# B&R Automation Studio project 305841_E00002_0 (part 11)

#### GAProcIO.fun - Exported functions and function blocks
```iecst
(********************************************************************
 * COPYRIGHT -- General Atomics
 ********************************************************************
 * Library: GAProcIO
 * File: GAProcIO.fun
 * Author: Administrator
 * Created: September 11, 2015
 ********************************************************************
 * Functions and function blocks of library GAAnalog
 ********************************************************************)

FUNCTION_BLOCK fbSclAlmAI (* Scale analog input and process alarms using the reference parameters *)
	VAR_INPUT
		_InInputStruct : REFERENCE TO sAnalogInput; (* structure representing the analog input to scale *)
		_InParamsStruct : REFERENCE TO sAnalogInputParams; (* structure representing the analog parameters *)
		_InSentinel : REAL; (* value to use if signal is invalid *) (* Set the scaling params and alm timer delays upon rising edge *) (* Must go low and high again to set again *)
		_InSetParams : BOOL := FALSE;
	END_VAR
	VAR
		SetParamsOS : BOOL := FALSE; (* set parameters one-shot *)
		rawAdj : REAL;
		almsRaw : UDINT; (* non-time delayed alarms *) (* deadband values, calculated from EU range and db pct *) (* pvs must rise above threshold by the corresponding value in order to be considered clear *)
		almRangeLoDbVal : REAL;
		almRangeHiDbVal : REAL;
		almLoLoDbVal : REAL;
		almLoDbVal : REAL; (* pvs must drop below threshold by the corresponding value in order to be considered clear *)
		almHiDbVal : REAL;
		almHiHiDbVal : REAL; (* alarm timers *)
		tmrAlmRangeLoOn : TON; (* on delay timers *)
		tmrAlmLoLoOn : TON;
		tmrAlmLoOn : TON;
		tmrAlmRangeHiOn : TON;
		tmrAlmHiOn : TON;
		tmrAlmHiHiOn : TON;
		tmrAlmRangeLoOff : TOF; (* off delay timers *)
		tmrAlmLoLoOff : TOF;
		tmrAlmLoOff : TOF;
		tmrAlmRangeHiOff : TOF;
		tmrAlmHiOff : TOF;
		tmrAlmHiHiOff : TOF;
		fbNoiseFilter : fbLpFilter; (* filter the scaled value *)
	END_VAR
END_FUNCTION_BLOCK

FUNCTION_BLOCK fbLpFilter (* Low pass filter *)
	VAR_INPUT
		_InPassThru : BOOL := FALSE; (* filter coefficient *) (* Value between 0 and 1, not inclusive of 1. *) (* K=0 no filtering, K=0.9999 lots of filtering *)
		_InK : REAL := 0.0;
		_InVal : REAL; (* input value *)
	END_VAR
	VAR_OUTPUT
		_OutFilteredVal : REAL; (* filtered value output  *)
	END_VAR
	VAR
		lastOut : REAL;
		firstScanOS : BOOL := FALSE;
		KChecked : REAL := 0.0;
	END_VAR
END_FUNCTION_BLOCK

FUNCTION_BLOCK fbProcDI (* process DI *)
	VAR_INPUT
		_InInputStruct : REFERENCE TO sDigitalInput; (* structure representing the digital input to process *)
		_InParamsStruct : REFERENCE TO sDigitalInputParams; (* structure representing the digital input parameters *)
		_InSentinel : BOOL := FALSE; (* value to use if signal is invalid *) (* Set the params and alm timer delays upon rising edge *) (* Must go low and high again to set again *)
		_InSetParams : BOOL := FALSE;
	END_VAR
	VAR
		SetParamsOS : BOOL := FALSE; (* set parameters one-shot *)
    value : BOOL;
    valueDly : BOOL;
    almsRaw : UDINT;
    prevParams : sDigitalInputParams; (* previous params -- used for auto param update *)
    paramSize : UDINT := 0;
    cmpResult : DINT;
		tmrOn : TON;
		tmrAlmLoOn : TON;
		tmrAlmHiOn : TON;
		tmrOff : TOF; (* non-time delayed alarms *)
		tmrAlmLoOff : TOF;
		tmrAlmHiOff : TOF;
	END_VAR
END_FUNCTION_BLOCK

FUNCTION_BLOCK fbProcPB
	VAR_INPUT
    _InPBIn : BOOL := FALSE;
    _InPBClear : BOOL := FALSE; (* Force state to be cleared *)
		_InPBType : eGAPIO_PB_BEHAVIOR_TYPE := GAPIO_PBBT_MOMENTARY;
		_InPulseTime : TIME := T#500ms;
	END_VAR
	VAR_OUTPUT
		_OutState : BOOL := FALSE;
	END_VAR
	VAR
		pressOS : BOOL := FALSE;
		state : BOOL := FALSE;
		tmrPulse : TON;
	END_VAR
END_FUNCTION_BLOCK
```

### Library Logical/Libraries/GAMpMotion (IEC) - Mapp Motion Helper Functions

#### Types.typ
```iecst
TYPE
  eGAMOT_HOME_FB_STATUS :
    (
    GAMOT_HMFBS_NOT_ACTIVE := 0,
    GAMOT_HMFBS_ENABLED := 1,
    GAMOT_HMFBS_HOMING := 2,
    GAMOT_HMFBS_HOMED := 3,
    GAMOT_HMFBS_ERR_START_STATE := -1, (* must be in disabled or standstill to start *)
    GAMOT_HMFBS_ERR_HOMING := -2 (* error occured during homing *)
  ) := GAMOT_HMFBS_NOT_ACTIVE;

  eGAMOT_AXIS_STATE_MACHINE_STATE :
    (
    (* axis state constants *)
    (* states which dont't issue move commands *)
    GAMOT_ASMS_INITIAL := 0, (*constant for an undefined state. Also used for initial state *)
    GAMOT_ASMS_IGNORE := 1, (*constant for ignore state *)
    GAMOT_ASMS_VALID_CHECK := 2, (*constant for invalid state *)
    GAMOT_ASMS_DISABLED := 3, (*constant for the disabled state *)
    GAMOT_ASMS_ENABLED := 4, (*constant for a waiting while powered *)
    GAMOT_ASMS_HOME_REQ := 5, (*constant for the state in which the axis home was requested *)
    GAMOT_ASMS_HOMING := 6, (*constant for the state in which the axis is being referenced *)
    GAMOT_ASMS_HOMED := 7, (*constant for the state in which the axis is referenced *)
    GAMOT_ASMS_CHK_RESTORE_POS := 8, (* constant for Init Endless Position State *)
    GAMOT_ASMS_RESTORE_POS := 9, (* constant for Init Endless Position Error State *)
    GAMOT_ASMS_ERROR_STOP := 10, (*constant for function block error stop state *)
    GAMOT_ASMS_ERROR_DRVRSTWAIT := 11, (*constant for axis error drive reset wait state *)
    GAMOT_ASMS_ERROR_DISABLE := 12, (*constant for axis error drive reset wait state *)
    GAMOT_ASMS_ERROR_DRVRST:= 13, (*constant for axis error drive reset state *)
    (* states which are stop moves *)
    GAMOT_ASMS_HALT := 20, (*constant for the state in which motion is halted *)
    GAMOT_ASMS_STOP := 21, (*constant for the state in which motion is stopped, awaiting stop reset req *)
    GAMOT_ASMS_STOP_RESET := 22, (*constant for the state in which movements are stopped after stop reset req received *)
    GAMOT_ASMS_HALT_DISABLE := 23, (* constant for the state which stops the axes before disabling *)
    (* states which are velocity  moves *)
    GAMOT_ASMS_JOG := 31, (*constant for the state in which jogging movement is executed *)
    GAMOT_ASMS_JOGPOSLIMIT := 32, (*constant for the state in which jogging positive limit movement is executed *)
    GAMOT_ASMS_JOGNEGLIMIT := 33, (*constant for the state in which jogging positive limit movement is executed *)
    (* states which are velocity moves *)
    GAMOT_ASMS_MOVE_VELOCITY := 41, (* constant for the state in which a movement with a defined velocity is executed *)
    (* states which are relative moves *)
    GAMOT_ASMS_MOVE_RELATIVE := 51, (*constant for the state in which a movement with defined distance is executed*)
    (* states which are absolute moves *)
    GAMOT_ASMS_MOVE_ABSOLUTE := 61, (*constant for the state in which a movement to defined position is executed *)
    (* states related to coordinated moves *)
    GAMOT_ASMS_ENGAGED_AS_SLAVE := 71, (* geared or cammed to a master axis (coordinated slave) *)
    GAMOT_ASMS_DISENGAGE_AS_SLAVE := 72 (* disengaging from a master axis (coordinated slave) *)
  ) := GAMOT_ASMS_INITIAL;

  eGAMOT_MOVE_DESIGNATION :
    ( (* Move Designation *)
    (* Be careful about changing values -- HMI ramifications *)
    (* Values support bit packed int *)
    GAMOT_MD_UNKNOWN                := -1, (* no HMI selection *)
    GAMOT_MD_NO_MOVE_COMMANDED      := 16#00,
    GAMOT_MD_JOG_VELOCITY_UP_FWD    := 16#01,
    GAMOT_MD_JOG_VELOCITY_DOWN_REV  := 16#02,
    GAMOT_MD_JOG_LIMIT_UP_FWD       := 16#04,
    GAMOT_MD_JOG_LIMIT_DOWN_REV     := 16#08,
    GAMOT_MD_VELOCITY               := 16#10,
    GAMOT_MD_RELATIVE               := 16#20,
    GAMOT_MD_ABSOLUTE               := 16#40,
    GAMOT_MD_COORDINATED            := 16#80
  ) := GAMOT_MD_NO_MOVE_COMMANDED;

  sMot_PositionLimits : STRUCT (* axis travel limits. *)
    (* This is a separate structure from move params so instances can
    efficiently be made permanent variables *)
    PositionLimitPos : LREAL;
    PositionLimitNeg : LREAL;
  END_STRUCT;

  sMot_HmiAxisReqs : STRUCT
    (* Move or motion related requests *)
    (* NOTE: BE CAREFUL about changes and reordering -- HMI and memcopy/memset ramifications *)
    (* Boolean reqs are cleared with memset so adding/removing/moving may be problematic *)
    (* NOTE: Do not add bool reqs before moveReq that should be cleared while in safe/emo modes. *)
    _beginResetSection : BOOL := FALSE;
    moveReq : BOOL := FALSE;
    haltReq : BOOL := FALSE;
    stopReq : BOOL := FALSE;
    homeSetZeroReq : BOOL := FALSE;
    homeSetOffsetReq : BOOL := FALSE;
    homeSetPosReq : BOOL := FALSE;
    enableReq : BOOL := FALSE;
    disableReq : BOOL := FALSE;
    manBrakeRelReq : BOOL := FALSE;
    clearManBrakeRelReq : BOOL := FALSE;
    offsetShiftReq : BOOL := FALSE; (* shift slave pos on the slave axis, shift value in slave units *)
    offsetShiftToMasterPosReq : BOOL := FALSE; (* shift slave position by axis offset in slave units *)
    phaseShiftReq : BOOL := FALSE; (* shift master pos on the slave axis, shift value in master units *)
    gearInReq : BOOL := FALSE;
    camInReq : BOOL := FALSE;
    disengageSlaveReq : BOOL := FALSE; (* Disengage cam and gear *)
    _endResetSection : BOOL := FALSE;
    (* NOTE: Do not add bool reqs after disengageSlaveReq that should be cleared in safe/emo modes.  HMI and memcopy/memset ramifications. *)
    (* Other requests *)
    (* NOTE: Do not add bool reqs before setPositionLimitsReq that should be cleared while in emo mode. *)
    (* Separate the below requests after disengageSlaveReq so they can be considered while in safe mode. *)
    (* These are things that can be done while in safe mode, but the ones above are cleared while in safe.*)
    setPositionLimitsReq : BOOL := FALSE;
    stopResetReq : BOOL := FALSE;
    errorResetReq : BOOL := FALSE;
    driveResetReq : BOOL := FALSE;
    axisNo : USINT := 0; (* convenience axis number this structure corresponds to *)
    (* gear in related *)
    gearRatioNumerator : DINT := 1000; (* gear factor of the slave / measurment resolution of the slave *)
    gearRatioDenominator : DINT := 1000; (* gear factor of the master / measurment resolution of the master *)
    (* shift related *)
    shiftOverMasterDistance : BOOL := FALSE; (* H: Perofrm shift over specified master distance Use mcPROFBASE_MASTER_DISTANCE and shiftProfileDistance *)
    shiftType : SINT := 0; (* based on HMI radio buttons. 0: Relative, 1: Abs *)
    shiftDistance : LREAL := 0.0; (* phase/offset shift distance *)
    shiftProfileDistance : LREAL := 0.0; (* distance master moves during a shift *)
    (* cam related *)
    camId : UINT;
    camMasterOffset : LREAL := 0.0; (* gear factor of the slave / measurment resolution of the slave *)
    camSlaveOffset : LREAL := 0.0; (* gear factor of the master / measurment resolution of the master *)
    homePosition : LREAL := 0.0;
    positionLimits : sMot_PositionLimits;
    moveDesignation : eGAMOT_MOVE_DESIGNATION := GAMOT_MD_NO_MOVE_COMMANDED;
    (* HMI move req *)
    (* BE CAREFUL ABOUT MOVING/DELETING/ADDING/CHANGING MEMORY between Direction and MaxJerk *)
    (* MAY NEED TO ADJUST fgProcessHmiMoveReq instruction in GaMpMotion library *)
    (* These move params are copied to/from the HMI move req structure using memcpy *)
    _startParamCopy : BOOL := FALSE;
    Direction : McDirectionEnum := mcDIR_UNDEFINED; (* direction for commanded movements*)
    Distance : LREAL := 0.0; (* distance for move Commands *)
    Position : LREAL := 0.0; (* target position for home or the motion *)
    Velocity : REAL := 0.0; (* velocity for move Commands *)
    Acceleration : REAL := 1.0; (* acceleration for commanded movements *)
    Deceleration : REAL := 1.0; (* deceleration for commanded movements *)
    MaxJerk : REAL := 0.0; (* deceleration for commanded movements *)
    _endParamCopy : BOOL := FALSE;
    (* NOTE: BE CAREFUL ABOUT MOVING/DELETING/ADDING/CHANGING MEMORY between direction and MaxJerk *)
  END_STRUCT;

  sMot_PermissiveCheck : 	STRUCT (* used to halt/stop if out of allowable range or due to permissive *)
    (* 24 byte structure *)
    PermissiveHaltNeg : BOOL; (* byte 0 *)
    PermissiveHaltPos : BOOL; (* byte 1 *)
    CheckFailed : BOOL; (* byte 2 *)
    RangeLimitNeg : BOOL; (* byte 3 *)
    RangeLimitPos : BOOL; (* byte 4 *)
    spareBytes : ARRAY[0..2] OF BYTE; (* bytes 5-7 *)
    StartPosition : LREAL; (* byte 8-15 *)
    EstStoppingDistance : LREAL; (* byte 16-23 *)
  END_STRUCT;

  sMot_AxisStatus : 	STRUCT  (* drive state structure from MC_ReadStatus *)
    (* MpAxisBasic related *)
    IsCommuncationReady : BOOL := FALSE; (* MpAxisBasic is ready to communicate *)
    IsReadyToPowerOn : BOOL := FALSE; (* MpAxisBasic is ready for operation *)
    (* digital input status *)
    IsAtHomingSwitch : BOOL := FALSE;
    IsAtPositiveLimitSwitch : BOOL := FALSE;
    IsAtNegativeLimitSwitch : BOOL := FALSE;
    IsTrigger1Active : BOOL := FALSE;
    IsTrigger2Active : BOOL := FALSE;
    IsDriveEnableActive : BOOL := FALSE;
    (* general status *)
    IsInSimulation : BOOL := FALSE; (* Axis is operating in simulaiton mode *)
    IsPoweredOn : BOOL := FALSE;  (* axis is swtiched on/enabled *)
    IsTorqueLimitReady : BOOL := FALSE;
    IsBrakeManuallyReleased : BOOL := FALSE;
    IsHomed : BOOL := FALSE; (* axis is referenced *)
    IsJogging : BOOL := FALSE; (* performing movement *)
    IsAtJogLimit : BOOL := FALSE; (* the axis has reached one of two position limits *)
    IsAtTorqueLimit : BOOL := FALSE; (* the axis limit is active *)
    IsInVelocity : BOOL := FALSE; (* axis is running with a defined velocity *)
    IsInPosition : BOOL := FALSE; (* axis has acheived the desired position *)
    IsMoveActive : BOOL := FALSE; (* movement is active *)
    IsMoveDone : BOOL := FALSE; (* move complete *)
    IsStopped : BOOL := FALSE; (* axis is stopped *)
    (* auto-tune related *)
    IsAutoTuneDone : BOOL := FALSE;
    AutoTuneQuality : REAL := 0.0;
    (* general status values and structures *)
    SafeMotionDiagCode : UINT; (* from Safety Controller safe motion instruction *)
    Velocity : REAL:= INVALID_SENTINEL_REAL; (* actual axis velocity *)
    Position : LREAL:= INVALID_SENTINEL_LREAL; (* actual axis position. Includes MOD to keep value within a period value *)
    DrivePosition : LREAL := INVALID_SENTINEL_LREAL; (* actual axis position. Does not includes MOD so period is ignored *)
    CalculatedPosition1 : LREAL:= INVALID_SENTINEL_LREAL; (* calculated position -- axis specific *)
    CalculatedPosition2 : LREAL:= INVALID_SENTINEL_LREAL; (* calculated position -- axis specific *)
    CalculatedPosition3 : LREAL:= INVALID_SENTINEL_LREAL; (* calculated position -- axis specific *)
    (* Values to see progress of a move *)
    MoveStartPos : LREAL := INVALID_SENTINEL_LREAL;
    MoveEndPos : LREAL := INVALID_SENTINEL_LREAL;
    MoveDistanceRemaining : LREAL := 0.0;
    MoveDistanceComplete : LREAL := 0.0;
    StartupCount : UDINT := 0; (* number of times the drive was started since last PLC start *)
    PlcOpenState : McAxisPLCopenStateEnum;
    networkCommState : McCommunicationStateEnum;
    AxisDiagnostics : MpAxisDiagExtType;
    LibraryInfo : McLibraryInfoType;
    (* coupling related *)
    HasCoordinatedSlave : BOOL := FALSE;
    IsGearInSync : BOOL := FALSE; (* slave is in sync with the master *)
    IsGearInCompensation : BOOL := FALSE; (* slave is in compensation with the master *)
    IsCamInSync : BOOL := FALSE; (* slave is in sync with the master *)
    IsCamEndOfProfile : BOOL := FALSE; (* Pulsed output indicating cyclic end of cam *)
    IsCoordOffsetShiftStarted : BOOL := FALSE;
    IsCoordOffsetShiftAttained : BOOL := FALSE;
    IsCoordPhaseShiftStarted : BOOL := FALSE;
    IsCoordPhaseShiftAttained : BOOL := FALSE;
    CamStatus : McCamInStatusEnum;
    CoordActualOffsetShift : LREAL := 0.0; (* current shift of the slave *)
    CoordActualPhaseShift : LREAL := 0.0; (* current shift of the master axis *)
  END_STRUCT;

  sMot_MoveParameters : 	STRUCT  (*parameter structure*)
    (* NOTE: BE CAREFUL about changes and reordering -- HMI and memcopy ramifications *)
    (* put the permissive stuff at the beginning, so the move parameter updates to the *)
    (* MpAxisBasic instruction deal with contiguous memory *)
    PosMovePermissive : BOOL := FALSE; (* byte 0 only allow forward moves when high *)
    NegMovePermissive : BOOL := FALSE; (* byte 1 only allow reverse moves when high *)
    EnableTorqueLimit : BOOL := FALSE; (* byte 2 Limit torque for accel/decel *)
    EnableTorqueLimitPrev : BOOL := FALSE;  (* byte 3 prev value to detect change *)
    HaltOnSlaveDisengage : BOOL := FALSE; (* byte 4 if set, issue a halt when axis is disengaged *)
    spareBytes5_7 : ARRAY[0..2] OF BYTE; (* bytes 5-7 *)
    PermissiveCheck : sMot_PermissiveCheck; (* 24 byte structure. bytes 8-31 permissive and range check bits *)
    VelocityMin : REAL := 0.001; (* bytes 32-35 min and max allowed velocity *)
    VelocityMax : REAL := 100.0; (* bytes 36-39 *)
    AccelMin : REAL := 0.001; (* bytes 40-43 min and max allowed acceleration *)
    AccelMax : REAL := 100.0; (* bytes 44-47 *)
    DecelMin : REAL := 0.001; (* bytes 48-51 min and max allowed deceleration *)
    DecelMax : REAL := 100.0; (* bytes 52-55 *)
    _beginHmiSection : BOOL := FALSE;
    (* HMI move req related *)
    (* BE CAREFUL ABOUT MOVING/DELETING/ADDING/CHANGING MEMORY between Direction and MaxJerk
    (* and between Direction to the end of the structure.*)
    (* MAY NEED TO ADJUST fgProcessHmiAxisReq instruction in GaMpMotion library *)
    (* These move params are copied to/from the HMI move req structure using memcpy *)
    (* use MC enum for direction *)
    (* mcPOSITIVE_DIR = 0, mcNEGATIVE_DIR = 1, mcDIR_SHORTEST_WAY = 3, mcDIR_UNDEFINED = 9, for other values, see docs *)
    Direction : McDirectionEnum := mcDIR_UNDEFINED; (* bytes 56-59 direction for commanded movements*)
    Distance : LREAL := 0.0; (* bytes 60-67 distance for move Commands*)
    Position : LREAL := 0.0; (* bytes 68-75 target position for the movement *)
    Velocity : REAL := 0.0; (* bytes 76-79 velocity for move Commands*)
    Acceleration : REAL := 1.0; (* bytes 80-83 acceleration for commanded movements*)
    Deceleration : REAL := 1.0; (* bytes 84-87 deceleration for commanded movements*)
    MaxJerk : REAL := 0.0; (* bytes 88-91 *)
    (* NOTE: BE CAREFUL ABOUT MOVING/DELETING/ADDING/CHANGING MEMORY between Direction and MaxJerk *)
    (* End Hmi Move Req *)
    _endHmiSection : BOOL := FALSE;
    HomeParams : MpAxisHomingType; (* parameters for referencing the axis*)
    JogParams : MpAxisJogType; (* parameters for jog command *)
    StopParams : MpAxisStopType; (* parameters for stop command *)
    TorqueLimitParams : MpAxisLimitLoadType; (* parameters for torque limit *)
    AutoTuneParams : MpAxisAutoTuneType; (* parameters for auto tuning *)
  END_STRUCT;

  sMot_CouplingParameters : 	STRUCT  (* coupling parameter structure*)
    CouplingPermissive : BOOL := FALSE; (* axis allowing itself to be coupled as a slave *)
    GearInReq : BOOL := FALSE; (* Set to request gear coupling *)
    GearOutReq : BOOL := FALSE; (* Set to request gear decoupling *)
    CamInReq : BOOL := FALSE; (* Set to request cam coupling *)
    CamOutReq : BOOL := FALSE; (* Set to request cam decoupling *)
    OffsetShiftReq : BOOL := FALSE;(* Generate an offset shift in the position of the slave on the slave axis *)
    PhaseShiftReq : BOOL := FALSE; (* Geneate a phase shift in the position of the master on the slave axis *)
    SlaveAxisNo : USINT := 0; (* default to 0 so setting a value can be detected *)
    (* CAUTION
    mem compare and mem copy are used for these values when dealing with run time value changes.
    Be very careful about where you add values. For example, changes to values in the gearin section will
    cause a gearin update *)
    (* Gear In params *)
    _beginGearInSection : BOOL := FALSE;
    GearInRatioNumerator : DINT := 1000; (* Gear factor of the slave / Measurement resolution of the slave *)
    GearInRatioDenominator : DINT:= 1000; (* Gear factor of the master / Measurement resolution of the master *)
    GearInMasterValueSource : McValueSrcEnum := mcVALUE_ACTUAL; (* Master position source *)
    GearInBufferMode : McBufferModeEnum := mcABORTING; (* mcABORTING is the only mode currently supported *)
    _endGearInSection : BOOL := FALSE;
    (* Offset / Phase shift params *)
    (* The values in the common section are common to gear in, cam, and shift *)
    _beginShiftCommonSection : BOOL := FALSE;
    ShiftAccelerationMax : REAL; (* if 0 limit for slave axis is used *)
    ShiftDecelerationMax : REAL; (* if 0 limit for slave axis is used *)
    ShiftJerk : REAL := 0.0; (* non zero only supported with McProfGen *)
    ShiftProfileBaseMaxVelocity : REAL := 0.0; (* also use for cam adv paramm vel. 0.0: use max velocity master axis *)
    _endShiftCommonSection : BOOL := FALSE;
    _beginShiftSection : BOOL := FALSE;
    ShiftMode : McShiftModeEnum;
    ShiftProfileBase : McProfileBaseEnum;
    Shift : LREAL; (* shift distance *)
    ShiftVelocityMax : REAL;
    ShiftProfileDistance : LREAL;
    (* Zone params used with profile base mcXxx_ZONE *)
    ShiftZoneStartPosition : LREAL;
    ShiftZoneEndPosition : LREAL;
    ShiftZonePeriod : LREAL := 0.0; (* 0: period defined for the profile base is used *)
    _endShiftSection : BOOL := FALSE;
    _beginCamInSection : BOOL := FALSE;
    CamIsPeriodic : BOOL := TRUE; (* H: cam is performed periodically, L: cam is performed once *)
    CamId : UINT := 1; (* cam id used with CamIn *)
    CamMasterOffset : LREAL := 0.0;
    CamSlaveOffset : LREAL := 0.0;
    CamScalingMaster : DINT := 1000; (* Cam scaling factor for master *)
    CamScalingSlave : DINT := 1000; (* Cam scaling factor for scaling *)
    CamStartMode : McCamStartModeEnum;
    CamMasterValueSource : McValueSrcEnum := mcVALUE_ACTUAL; (* Master position source *)
    CamBufferMode : McBufferModeEnum := mcABORTING; (* mcABORTING is thye only mode currently supported *)
    _endCamInSection : BOOL := FALSE;
  END_STRUCT;

  sMot_AxisCommands : 	STRUCT  (*command structure for single and master axes*)
    MoveNotAllowed : BOOL:= TRUE; (* set if a requested move is not allowed, clear upon good request *)
    PlcSafetyEnable : BOOL := FALSE; (* PLC logic enable of SafeMC, via safety controller *)
    UpdateMoveParams : BOOL := FALSE; (* used to control the update bit to McAxisBasic when move params change *)
    EnableReq : BOOL:= FALSE; (* request enabling (powering on) the controller. *)
    DisableReq : BOOL:= FALSE; (* request disabeling (powering off) the controller *)
    EnableCmd : BOOL:= FALSE; (* enable (power on) the controller. Power off on false *)
    ReleaseBrakeReq : BOOL:= FALSE; (* request brake release if motor is off *)
    ClearReleaseBrakeReq : BOOL:= FALSE; (* clear brake release req *)
    ReleaseBrakeCmd : BOOL:= FALSE; (* release brake if motor is off *)
    HomeReq : BOOL:= FALSE; (* request setting of the reference position *)
    HomeCmd : BOOL:= FALSE; (* set the reference position *)
    MoveJogReq : BOOL:= FALSE; (* request jog move as long as is set. Direction set by MoveParameter.Direction *)
    MoveJogCmd : BOOL:= FALSE; (* jog (move) as long as is set. Direction set by MoveParameter.Direction *)
    MoveJogPositiveReq : BOOL:= FALSE; (* request jog move as long as is set. Stop at the software position limit *)
    MoveJogPositiveCmd : BOOL:= FALSE; (* jog (move) as long as is set. Stop at the software position limit *)
    MoveJogNegativeReq : BOOL:= FALSE; (* request jog move as long as is set. Stop at the software position limit *)
    MoveJogNegativeCmd : BOOL:= FALSE; (* jog (move) as long as is set. Stop at the software position limit *)
    MoveVelocityReq : BOOL:= FALSE; (* request move at a defined velocity *)
    MoveVelocityCmd : BOOL:= FALSE; (* move at a defined velocity *)
    MoveRelativeReq : BOOL:= FALSE; (* request move of a defined distance*)
    MoveRelativeCmd : BOOL:= FALSE; (* move a defined distance *)
    MoveAbsoluteReq : BOOL:= FALSE; (* request move to a defined position *)
    MoveAbsoluteCmd : BOOL:= FALSE; (* move to a defined position *)
    StopReq : BOOL:= FALSE; (* reqeust stop every active movement on the axis as long as is set *)
    StopCmd : BOOL:= FALSE; (* stop every active movement on the axis as long as is set *)
    StopResetReq : BOOL:= FALSE; (* set high to get out of STOPPED state *)
    HaltReq : BOOL:= FALSE; (* request stop every active movement on the axis *)
    HaltCmd : BOOL:= FALSE; (* stop every active movement on the axis *)
    DriveResetReq : BOOL:= FALSE; (* request drive reset *)
    DriveResetCmd : BOOL:= FALSE; (* drive reset command *)
    ErrorResetReq : BOOL:= FALSE; (* Request exit from Error Reset Wait *)
  END_STRUCT;

(*
  sMot_Error : 	STRUCT  (*error structure
    FBError : BOOL; (*an error occurred in a FB
    AxisError : BOOL; (*an axis error has occurred
    AxisWarning : BOOL; (*an axis warning has occurred
    AxisErrorStop : BOOL; (*axis is in ErrorStop state
    AcknowledgeAllReq : BOOL; (*user alarm acknowledge - ack all alarms
    AcknowledgeReq : BOOL; (*user alarm acknowledge
    AxisErrorCount : UINT; (*number of active axis errors
    AxisWarningCount : UINT; (*number of active axis warinings
    FBErrorCount : UINT; (*number of active function block errors
    ErrorText : ARRAY[0..3]OF STRING[79]; (*description of first active error or warning
    DateObjectName : STRING[32]; (* Name of rrror text table data object
  END_STRUCT;
*)
(*
  sMot_FbStatus : 	STRUCT
    Active : BOOL;
    Error : BOOL;
    UpdateDone : BOOL;
    CommandBusy : BOOL;
    CommandAborted : BOOL;
    ExecutingCommand : MpAxisExecutingCmdEnum;
    StatusId : MpAxisErrorEnum; (* axis error
    StatusSeverity : MpComSeveritiesEnum;
    StatusCode : UINT;
    InternalId : DINT; (* status number of the implementation specific library
    InternalSeverity: MpComSeveritiesEnum; (* type of info returned by status id
    InternalFacility: MpComFacilitiesEnum; (* system responsible for the error
    InternalCode: UINT; (* decode value of Status ID -- error number is left over
  END_STRUCT;
*)
  sMot_Axis : 	STRUCT  (*substructure for single and master axes*)
    Ignore : BOOL := TRUE; (* when set, some software routines ignore this axis. Default to set so dummy axis is ignored *)
    ForceSetRef : BOOL := TRUE; (* force the operator to have to re-reference the axis *)
    StartupHomeOk : BOOL := FALSE; (* axis can home itself after startup *)
    isAxisVirtual : BOOL := FALSE; (* axis is virtual if true and motion commands are not allowed *)
    isAxisEndless : BOOL := FALSE; (* axis has no physical limits *)
    isAxisInverter : BOOL := FALSE; (* axis is an inverter in motion control mode *)
    AxisNo : USINT := GAMOT_ASMS_INITIAL; (* default to initial so setting a value can be detected *)
    SMState : eGAMOT_AXIS_STATE_MACHINE_STATE := 0; (* enumeration managed by the state machine *)
    AxisObj : McAxisType ; (* reference to global axis object (i.e. the drive) *)
    SlaveAxisObj : McAxisType ; (* reference to global axis object (i.e. the drive) *)
    Status : sMot_AxisStatus; (* status of the slave axis *)
    StatusSlave : sMot_AxisStatus; (* status of the slave axis *)
    MoveParameters : sMot_MoveParameters; (*parameter structure*)
    MoveParametersPrev : sMot_MoveParameters;  (* detect changes *)
    CouplingParameters : sMot_CouplingParameters;
    CouplingParametersPrev : sMot_CouplingParameters; (* detect changes *)
    Commands : sMot_AxisCommands; (*command structure for single and master axes*)
    fbMpAxisBasic : MpAxisBasic;
    fbReadDrivePos : MC_BR_ReadCyclicPosition;
    fbUpdateBFbParams : fbUpdateBasicParams;
    fbGearIn : MC_GearIn;
    fbGearOut : MC_GearOut;
    fbOffsetShift : MC_BR_Offset;
    fbPhaseShift : MC_BR_Phasing;
    fbCalcCam : MC_BR_CalcCamFromSections;
    fbCalcPoints : MC_BR_CalcPointsFromCam;
    fbCamPrepare : MC_BR_CamPrepare;
    fbCamIn : MC_CamIn;
    fbCamOut : MC_CamOut;
    fbCheckRestorePos : MC_BR_CheckRestorePositionData;
  END_STRUCT;

  sMot_GlobalCommands : 	STRUCT  (*command structure for global axis commands*)
    EnableReq : BOOL := FALSE; (* Request all axes be enabled (switched on) *)
    DisableReq : BOOL := FALSE; (* Request all axes be disabled (switched off) *)
    HaltReq : BOOL := FALSE; (* Request to halt as long as is set *)
    StopReq : BOOL := FALSE; (* Request to stop as long as is set *)
    ErrorAcknowledge : BOOL := FALSE; (*reset active errors*)
  END_STRUCT;

END_TYPE
```

#### GAMpMotion.fun
```iecst
FUNCTION_BLOCK fbHomeAbsSeq
  VAR_INPUT
    _I_Enable   : BOOL;
    _I_Axis     : REFERENCE TO sMot_Axis;
    _I_Position : LREAL;
  END_VAR
  VAR_OUTPUT
    _O_Done  : BOOL;
    _O_Busy  : BOOL;
    _O_Error : BOOL;
    _O_Homed : BOOL;
    _O_State : eGAMOT_HOME_FB_STATUS;
  END_VAR
  VAR
    enableOS : BOOL;
  END_VAR
  VAR CONSTANT
  END_VAR
END_FUNCTION_BLOCK

FUNCTION_BLOCK fbProcessHmiAxisReq   (* Process axis requests from HMI and populate axis structure(s) *)
  VAR_INPUT
    _I_HmiAxisReq : REFERENCE TO sMot_HmiAxisReqs;
    _I_Axis : REFERENCE TO sMot_Axis;
    _I_SlaveAxis : REFERENCE TO sMot_Axis;
    _I_AxisPositionLimits : REFERENCE TO sMot_PositionLimits;
    _I_ToleranceZeroDepth : LREAL := 0.001;
  END_VAR

  VAR
    pHmi :  UDINT;
    pMoveParams :  UDINT;
    size :  UDINT;
    nxtAddr :  UDINT;
    fbHomeSeq : fbHomeAbsSeq;
  END_VAR

END_FUNCTION_BLOCK

FUNCTION_BLOCK fbUpdateBasicParams
  VAR_INPUT
    _I_Axis : REFERENCE TO sMot_Axis;
  END_VAR
  VAR_IN_OUT
    _IO_MpParams : MpAxisBasicParType; (* Mapp Motion move param structure *)
	END_VAR
  VAR
		updateOS :  BOOL := FALSE;
    result : DINT;
    pParamsStart :  UDINT := 0;
    pParamsEnd :  UDINT := 0;
    pParamsPrev :  UDINT := 0;
    size : UDINT := 0;
    nxtAddr : UDINT;
  END_VAR
END_FUNCTION_BLOCK

FUNCTION fctCalcAbsHomeOffset : LREAL (* Return encoder offset for absolute home mode *)
  VAR_INPUT
    _I_CurrentPos : LREAL;
    _I_DesiredPos : LREAL;
    _I_SetZeroOffset : LREAL := 0.0;
  END_VAR
END_FUNCTION

FUNCTION fctCheckEqCamInParams : BOOL (*Return true if the two structures are equal*)
	VAR_INPUT
		_I_ParamsA : REFERENCE TO sMot_CouplingParameters;
		_I_ParamsB : REFERENCE TO sMot_CouplingParameters;
	END_VAR
	VAR
    pParamsStart :  UDINT := 0;
    pParamsEnd :  UDINT := 0;
    pParamsPrev :  UDINT := 0;
    size : UDINT := 0;
    result : UDINT;
	END_VAR
END_FUNCTION

FUNCTION fctCheckEqGearInParams : BOOL (*Return true if the two structures are equal*)
	VAR_INPUT
		_I_ParamsA : REFERENCE TO sMot_CouplingParameters;
		_I_ParamsB : REFERENCE TO sMot_CouplingParameters;
	END_VAR
	VAR
    pParamsStart :  UDINT := 0;
    pParamsEnd :  UDINT := 0;
    pParamsPrev :  UDINT := 0;
    size : UDINT := 0;
    result : UDINT;
	END_VAR
END_FUNCTION

FUNCTION fctCheckEqMoveParams : BOOL (*Return true if the two structures are equal*)
	VAR_INPUT
		_I_ParamsA : REFERENCE TO sMot_MoveParameters;
		_I_ParamsB : REFERENCE TO sMot_MoveParameters;
	END_VAR
	VAR
		size : UDINT;
		result : DINT;
	END_VAR
END_FUNCTION

FUNCTION fctCheckEqShiftParams : BOOL (*Return true if the two structures are equal*)
	VAR_INPUT
		_I_ParamsA : REFERENCE TO sMot_CouplingParameters;
		_I_ParamsB : REFERENCE TO sMot_CouplingParameters;
	END_VAR
	VAR
    pParamsStart :  UDINT := 0;
    pParamsEnd :  UDINT := 0;
    pParamsPrev :  UDINT := 0;
    size : UDINT := 0;
    result : UDINT;
	END_VAR
END_FUNCTION

FUNCTION fctClearMotionCommands : BOOL (*Clear command bits in the _IO_sMot_Command parameter if the bit in the eMOT_AXIS_CMD_MASK input mask is clear*)
	VAR_INPUT
		_I_CmdMask : DINT := 0; (* command bit mask -- do not clear the commands corresponding to set bits*)
	END_VAR
	VAR_IN_OUT
		_IO_Commands : sMot_AxisCommands; (* commands structure -- clear all cmd bits, except those with the mask bit set *)
	END_VAR
END_FUNCTION

FUNCTION fctClearMotionRequests : BOOL (*Clear request bits in the _IO_sMot_Command parameter if the bit in the eMOT_AXIS_CMD_MASK input mask is clear*)
  VAR_INPUT
    _I_ReqMask : DINT := 0; (*request bit mask -- do not clear the requests corresponding to set bits*)
  END_VAR
  VAR_IN_OUT
    _IO_Commands : sMot_AxisCommands; (*commands structure -- clear all req bits, except those with the mask bit set *)
  END_VAR
END_FUNCTION

FUNCTION fctCopyAxisStatus : BOOL
  VAR_INPUT
    _I_SrcStatus : REFERENCE TO sMot_AxisStatus;
    _I_DestStatus : REFERENCE TO sMot_AxisStatus;
  END_VAR
  VAR
    (* result :  DINT; *)
    (* pSrc :  UDINT; *)
    (* pDest :  UDINT; *)
    (* size : UDINT; *)
    nxtAddr : DINT;
  END_VAR

END_FUNCTION

FUNCTION fctGetMpAxisInfo : BOOL (*Pack values stored in a MpAxisBasicInfoType structure into a sMot_AxisStatus structure*)
  VAR_INPUT
    _I_MpInfo : REFERENCE TO MpAxisBasicInfoType; (* packed Mapp Motion structure *)
  END_VAR
  VAR_IN_OUT
    _IO_UdtStatus : sMot_AxisStatus; (* input move params in a udt *)
  END_VAR
END_FUNCTION

FUNCTION fctPackMpAxisBasicParams : BOOL (*Pack values stored in a sMot_MoveParameter structure into a MpAxisBasicParType structure *)
  VAR_INPUT
    _I_UdtParams : REFERENCE TO sMot_MoveParameters; (* input move params in a udt *)
  END_VAR
  VAR_IN_OUT
    _IO_MpParams : MpAxisBasicParType; (* packed Mapp Motion structure *)
  END_VAR
END_FUNCTION
```

#### GAMpMotion.st
```iecst
// Given an referenced to an sMot_Axis structure, and
// a desired position, request an absolute move on the axis.
// This funciton block is intended to be called all the time,
// and perform the home when the enable input is set.  It allows
// easy monitoring of its outputs to see when homing is complete.
FUNCTION_BLOCK fbHomeAbsSeq
  IF NOT _I_Enable THEN
    // Not enabled. Clear OS, clear outputs and leave
    enableOS := FALSE;
    _O_Busy := FALSE;
    _O_Done := FALSE;
    _O_Error := FALSE;
    _O_Homed := FALSE;
    _O_State := GAMOT_HMFBS_NOT_ACTIVE;
    RETURN;
  ELSIF _I_Enable AND NOT enableOS THEN
    // Enable rising edge ... Set the OS and update the fb outputs.
    // Axis needs to be in disable or standstill states to start homing.
    // If not, return an error, but if so, then set the mode and position and requst
    // homing.

    // Set OS
    enableOS := TRUE;

    IF _I_Axis.Status.PlcOpenState <> mcAXIS_DISABLED AND _I_Axis.Status.PlcOpenState <> mcAXIS_STANDSTILL THEN
      // Not disabled or standstill... This is an error, must be here to home.
      _O_Busy := FALSE;
      _O_Done := TRUE;
      _O_Error := TRUE;
      _O_Homed := FALSE;
      _O_State := GAMOT_HMFBS_ERR_START_STATE;
    ELSE
      // In standstill or disabled... Okay to start homing.
      // This is the first pass, so set up home cmd.
      // Set the position here on the first scan, and then not again ...
      // Don't want an updated position passed into the fb as a result of homing
      // to confuse things.
      // If the axis is virtual, use direct, otherwise use absolute
      IF _I_Axis.isAxisVirtual THEN
          // The virtual axis case
        _I_Axis.MoveParameters.HomeParams.Mode := mcHOMING_DIRECT;
      ELSE
        //. The non-virtual axis case
        _I_Axis.MoveParameters.HomeParams.Mode := mcHOMING_DIRECT;
      END_IF;

      _I_Axis.MoveParameters.HomeParams.Position := _I_Position;
      _I_Axis.Commands.HomeReq := TRUE;
      _O_Busy  := TRUE;
      _O_Done  := FALSE;
      _O_Error := FALSE;
      _O_Homed := FALSE;
      _O_State := GAMOT_HMFBS_ENABLED;
    END_IF;

  ELSE
    // While Enabled (after rising edge)
    IF _O_State = GAMOT_HMFBS_ENABLED AND
      (_I_Axis.Status.PlcOpenState = mcAXIS_HOMING OR
      _I_Axis.Status.AxisDiagnostics.ExecutingCommand = mcAXIS_CMD_HOMING) THEN
      // state is homing
      _O_Busy  := TRUE;
      _O_Done  := FALSE;
      _O_Error := FALSE;
      _O_Homed := FALSE;
      _O_State := GAMOT_HMFBS_HOMING;
    ELSIF _O_State = GAMOT_HMFBS_HOMING AND _I_Axis.Status.IsHomed AND
      (_I_Axis.Status.PlcOpenState = mcAXIS_DISABLED OR
      _I_Axis.Status.PlcOpenState = mcAXIS_STANDSTILL) THEN
      // Force to go thru the homing state, but now done (sucessfully homed)
      _O_Busy  := FALSE;
      _O_Done  := TRUE;
      _O_Error := FALSE;
      _O_Homed := TRUE;
      _O_State := GAMOT_HMFBS_HOMED;
    ELSIF _O_State = GAMOT_HMFBS_HOMING AND
      (_I_Axis.Status.AxisDiagnostics.StatusID.ID <> mcAXIS_NO_ERROR OR
      _I_Axis.Status.PlcOpenState = mcAXIS_ERRORSTOP) THEN
      // Force to go thru the homing state, but now done -- error case
      _O_Busy  := FALSE;
      _O_Done  := TRUE;
      _O_Error := TRUE;
      _O_Homed := FALSE;
      _O_State := GAMOT_HMFBS_ERR_HOMING;
    END_IF;
  END_IF;
END_FUNCTION_BLOCK

// If an axis request is made, copy the hmi values to the correct axis structure(s),
// and set the request in the axis command structure.
// NOTE: It is important to clear the HMI requests immediatly after acting on them.
// This is because the binding of the HMI is such that a high request will be set on
// whichever axis is selected. If a the operator changes the selected axis, the
// requst bit on the newly selected axis must not be set because the requst on the
// origianl axis was high.
FUNCTION_BLOCK fbProcessHmiAxisReq
  // If a halt or a stop request is made, make these priority.
  // Make sure the move request is cleared, so it does not get serviced,
  // and send the halt or stop, and clear the requests.
  IF _I_HmiAxisReq.stopReq OR _I_HmiAxisReq.haltReq THEN
    // Clear the move reqs
    _I_HmiAxisReq.moveReq := FALSE;
    _I_HmiAxisReq.moveDesignation := GAMOT_MD_NO_MOVE_COMMANDED;
    // Note the axis SM will handle the clearing of the axis.commands.reqs.
    // Send thru the requested stop or halt
    _I_Axis.Commands.StopReq:= _I_HmiAxisReq.stopReq;
    _I_Axis.Commands.HaltReq := _I_HmiAxisReq.haltReq;
    // reset the hmi requests
    _I_HmiAxisReq.stopReq := FALSE;
    _I_HmiAxisReq.haltReq := FALSE;
  END_IF;

  // Set permanent varialbe position limits if requested
  IF _I_HmiAxisReq.setPositionLimitsReq THEN
    // Clear the request
    _I_HmiAxisReq.setPositionLimitsReq := FALSE;
    // Set the retained limits to the requested values.
    _I_AxisPositionLimits.PositionLimitPos := _I_HmiAxisReq.positionLimits.PositionLimitPos;
    _I_AxisPositionLimits.PositionLimitNeg := _I_HmiAxisReq.positionLimits.PositionLimitNeg;
  END_IF;

  // Put the position, velocity, accel, decel and max jerk from the HMI axis request into the axis structures.
  // NOTE: Assume identical memory layout ... memcpy used
  // memcpy(dest, src, len);
  pHmi := ADR(_I_HmiAxisReq.Position);
  pMoveParams := ADR(_I_Axis.MoveParameters.Position);
  size:= ADR(_I_HmiAxisReq.MaxJerk) - ADR(_I_HmiAxisReq.Position) + SIZEOF(_I_HmiAxisReq.MaxJerk); // bytes of the hmi move req moved to the appropriate section of the axis move parameters
  nxtAddr := brsmemcpy(pMoveParams,pHmi,size);

  // Update coupling params if a slave axis is designated for this axis.
  // The slave need not be engaged. The engage/disengage, gear, and shfit requests are handled later.
  // These parameters are loaded from the HMI values here, ahead of the request, such that
  // an HMI change can be detected and acted on below (gear change for example).
  IF _I_Axis.CouplingParameters.SlaveAxisNo <> 0 THEN
    // Load the params. Use values from the HMI structure when available

    // *** Gear In Params
    _I_Axis.CouplingParameters.GearInRatioNumerator := _I_HmiAxisReq.gearRatioNumerator;
    _I_Axis.CouplingParameters.GearInRatioDenominator := _I_HmiAxisReq.gearRatioDenominator;
    _I_Axis.CouplingParameters.GearInMasterValueSource := mcVALUE_SET;
    _I_Axis.CouplingParameters.GearInBufferMode := mcABORTING;
    // Gear In,Offset Shift and Phase shift all use the slave accel/decel values,
    // so make sure the values are set in the coupling params structure
    _I_Axis.CouplingParameters.ShiftAccelerationMax := _I_SlaveAxis.MoveParameters.AccelMax; // slave accel. Set to 0.0 to use slave max
    _I_Axis.CouplingParameters.ShiftDecelerationMax := _I_SlaveAxis.MoveParameters.DecelMax; // slave decel. Set to 0.0 to use slave max
    _I_Axis.CouplingParameters.ShiftJerk := 0.0; // non-zero only supported with McProfGen
    _I_Axis.CouplingParameters.ShiftProfileBaseMaxVelocity := 0.0; // _I_Axis.MoveParameters.VelocityMax; // Allow master max velocity

    // *** Cam params
    // _I_Axis.CouplingParameters.CamIsPeriodic := FALSE; // TODO: Bring to UI
    _I_Axis.CouplingParameters.CamId := _I_HmiAxisReq.camId;
    // Allow different cams to have different scaling
    // This allows the cam tables to be in different units (degrees, % of motion, revs, etc) for example
    IF _I_Axis.CouplingParameters.CamId = 1 THEN // Placeholder to show the concept
      // Cam table in units of degrees, and resolution is 0.001 for both axes
      _I_Axis.CouplingParameters.CamScalingMaster := 1000;
      _I_Axis.CouplingParameters.CamScalingSlave := 1000;
    ELSE
      // Assume Cam table is in units of degrees, and resolution is 0.001 for both axes
      _I_Axis.CouplingParameters.CamScalingMaster := 1000;
      _I_Axis.CouplingParameters.CamScalingSlave := 1000;
    END_IF;
    // mcCAM_START_DIRECT: Start the cam using the current position of the master and slave.
    // Use the master offset to set how far into the cam until starting takes place
    // Slave offset is not used
    _I_Axis.CouplingParameters.CamStartMode := mcCAM_START_DIRECT;
    _I_Axis.CouplingParameters.CamMasterOffset := _I_HmiAxisReq.camMasterOffset;
    _I_Axis.CouplingParameters.CamSlaveOffset := _I_HmiAxisReq.camSlaveOffset;
    // TODO: Actual or set point??
    // _I_Axis.CouplingParameters.CamMasterValueSource := mcVALUE_ACTUAL;
    _I_Axis.CouplingParameters.CamMasterValueSource := mcVALUE_SET;
    _I_Axis.CouplingParameters.CamBufferMode := mcABORTING; (* mcABORTING is thye only mode currently supported *)

    // *** Shift & offset related values
    // accel, decel, jerk and base max vel set above
    _I_Axis.CouplingParameters.Shift := _I_HmiAxisReq.shiftDistance; // slave shift distance
    _I_Axis.CouplingParameters.ShiftVelocityMax := _I_SlaveAxis.MoveParameters.VelocityMax; // Use slave max velocity
    // use shift profile distance with mcPROFBASE_MASTER_DISTANCE profile base
    _I_Axis.CouplingParameters.ShiftProfileDistance :=  _I_HmiAxisReq.shiftProfileDistance; // master distance over which to perform the shift

  END_IF;

  IF _I_HmiAxisReq.moveReq THEN
    // A move request is made ...
    // The move paramaters will be set based on the HMI request values.
    // Note that the HMI requests specify a direction and a positive distance
    // for a relative move, but the axis SM uses a signed distance value.
    // For a relative move, convert the distance specification into a signed distance.
    IF _I_HmiAxisReq.moveDesignation = GAMOT_MD_RELATIVE AND _I_HmiAxisReq.Direction = mcDIR_POSITIVE THEN
      // Relative move in the positive direction.
      // Ensure distance is positive, and set the direction to undefined (not used)
      _I_Axis.MoveParameters.Distance := ABS(_I_HmiAxisReq.Distance);
      _I_Axis.MoveParameters.Direction := mcDIR_UNDEFINED;
    ELSIF _I_HmiAxisReq.moveDesignation = GAMOT_MD_RELATIVE AND _I_HmiAxisReq.Direction = mcDIR_NEGATIVE THEN
      // Relative move in the negative direction.
      // Ensure distance is negative, and set the direction to undefined (not used)
      _I_Axis.MoveParameters.Distance := -1.0 * ABS(_I_HmiAxisReq.Distance);
      _I_Axis.MoveParameters.Direction := mcDIR_UNDEFINED;
    ELSIF _I_HmiAxisReq.moveDesignation = GAMOT_MD_RELATIVE THEN
      // Relative move, but not positive or negative direction.
      // Don't move ... set distance to zero
      _I_Axis.MoveParameters.Distance := 0.0;
      _I_Axis.MoveParameters.Direction := mcDIR_UNDEFINED;
    ELSE
      // Not a relative move. Use the direction and distance as specified.
      _I_Axis.MoveParameters.Distance := _I_HmiAxisReq.Distance;
      _I_Axis.MoveParameters.Direction := _I_HmiAxisReq.Direction;
    END_IF;

    // Now set the move request based on the move designation
    // The move designaiton only holds a single value (duh!), so only
    // one of the following should evalutate to true
    // If direction is specified in move designaiton, it must match the selected direction
    _I_Axis.Commands.MoveJogReq := (
    ((_I_HmiAxisReq.moveDesignation = GAMOT_MD_JOG_VELOCITY_UP_FWD) AND (_I_HmiAxisReq.Direction = mcDIR_POSITIVE)) OR
    ((_I_HmiAxisReq.moveDesignation = GAMOT_MD_JOG_VELOCITY_DOWN_REV) AND (_I_HmiAxisReq.Direction = mcDIR_NEGATIVE))
    );
    _I_Axis.Commands.MoveJogPositiveReq := (_I_HmiAxisReq.moveDesignation = GAMOT_MD_JOG_LIMIT_UP_FWD) AND (_I_HmiAxisReq.Direction = mcDIR_POSITIVE);
    _I_Axis.Commands.MoveJogNegativeReq := (_I_HmiAxisReq.moveDesignation = GAMOT_MD_JOG_LIMIT_DOWN_REV) AND (_I_HmiAxisReq.Direction = mcDIR_NEGATIVE);
    _I_Axis.Commands.MoveVelocityReq := _I_HmiAxisReq.moveDesignation = GAMOT_MD_VELOCITY;
    _I_Axis.Commands.MoveRelativeReq := _I_HmiAxisReq.moveDesignation = GAMOT_MD_RELATIVE;
    _I_Axis.Commands.MoveAbsoluteReq := _I_HmiAxisReq.moveDesignation = GAMOT_MD_ABSOLUTE;
    // Move request and designation processed ...
    // Clear the move request and move designation so it is processed again if requested again.
    // The axis SM will handle the maintaining or clearing of the axis.commands.reqs.  Note the Velocity and Jog cmds are maintained until stopped.
    _I_HmiAxisReq.moveReq := FALSE;
    _I_HmiAxisReq.moveDesignation := GAMOT_MD_NO_MOVE_COMMANDED;
  END_IF;

  // Handle a coupling or decoupling (gear in or cam in) request.
  // Only allow coupling if a slave is designated and the slave allows it
  // Decouple on request as long as there is a slave designated.
  IF _I_Axis.CouplingParameters.SlaveAxisNo = 0 THEN
    // No slave designated
    // Clear the request
    _I_HmiAxisReq.gearInReq := FALSE;
    _I_HmiAxisReq.camInReq := FALSE;
  // Slave must be designated to get past this, so no need to keep checking
  ELSIF _I_SlaveAxis.Status.PlcOpenState = mcAXIS_SYNCHRONIZED_MOTION AND
        (_I_HmiAxisReq.disengageSlaveReq OR NOT _I_SlaveAxis.CouplingParameters.CouplingPermissive) THEN
    // Slave is coupled, but disengage slave request or coupling not allowed.
    // Turn off gearing, caming, block the engage reqs, and clear the disengage req
    _I_Axis.CouplingParameters.GearOutReq := TRUE;
    _I_Axis.CouplingParameters.CamOutReq := TRUE;
    _I_HmiAxisReq.gearInReq := FALSE;
    _I_HmiAxisReq.camInReq := FALSE;
    _I_HmiAxisReq.disengageSlaveReq := FALSE;
  ELSIF _I_HmiAxisReq.gearInReq AND _I_SlaveAxis.CouplingParameters.CouplingPermissive THEN
    // Gear in requested and allowed.
    // Turn on gearing and clear the requst
    _I_Axis.CouplingParameters.GearInReq := TRUE;
    _I_HmiAxisReq.gearInReq := FALSE;
    // make sure the cam req is cleared
    _I_Axis.CouplingParameters.CamInReq := FALSE;
  ELSIF _I_HmiAxisReq.camInReq AND _I_SlaveAxis.CouplingParameters.CouplingPermissive THEN
    // Cam in requested and allowed
    // Turn on caming and clear the requst
    _I_Axis.CouplingParameters.CamInReq := TRUE;
    _I_HmiAxisReq.camInReq := FALSE;
    // make sure the gear in req is cleared
    _I_Axis.CouplingParameters.GearInReq := FALSE;
  END_IF;

  // Handle a offset or phase shift request
  // Only one at a time, so both handled by this conditional
  // Cancel the reqs if the master isn't moving, or if the slave is not coordinated,
  // or if the shift amount is zero, or the profile (master) distance is being used but is set to zero,
  // or a phase or offset shift is in progress

  IF // master not moving or slave not coordinated
      NOT _I_Axis.Status.IsMoveActive OR
      NOT _I_Axis.Status.IsGearInSync OR
      // Zero relative shift distance requested
      ((_I_HmiAxisReq.offsetShiftReq OR _I_HmiAxisReq.phaseShiftReq) AND _I_HmiAxisReq.shiftType = 0 AND _I_HmiAxisReq.shiftDistance = 0.0) OR
      // zero out position offset to master, but position offset is zero
      (_I_HmiAxisReq.offsetShiftToMasterPosReq AND ABS(_I_SlaveAxis.Status.CalculatedPosition1) < _I_ToleranceZeroDepth) OR
      // master distance profile base and zero profile distance
      (_I_HmiAxisReq.shiftOverMasterDistance AND
       _I_HmiAxisReq.shiftProfileDistance = 0.0) OR
       // a shift is active
       _I_Axis.fbOffsetShift.ShiftStarted OR
       _I_Axis.fbPhaseShift.ShiftStarted THEN
    // Turn off shifting, block the shift reqs, and clear the end req
    _I_HmiAxisReq.offsetShiftReq := FALSE;
    _I_HmiAxisReq.offsetShiftToMasterPosReq := FALSE;
    _I_HmiAxisReq.phaseShiftReq := FALSE;
  ELSIF _I_HmiAxisReq.offsetShiftReq OR _I_HmiAxisReq.offsetShiftToMasterPosReq THEN
    // New offset request
    // The non request specific params in the coupling structure were set above.
    // Here we need to handle request specific stuff

    // Look at the shift type to determine absolute or relative
    IF _I_HmiAxisReq.shiftType = 0 OR _I_HmiAxisReq.offsetShiftToMasterPosReq THEN
      // relative
      _I_Axis.CouplingParameters.ShiftMode := mcSHIFT_RELATIVE_NO_RESET;
    ELSIF _I_HmiAxisReq.shiftType = 1 THEN
      // absolute
      _I_Axis.CouplingParameters.ShiftMode := mcSHIFT_ABSOLUTE_NO_RESET;
    ELSE // catch-all -- use relative
      _I_Axis.CouplingParameters.ShiftMode := mcSHIFT_RELATIVE_NO_RESET;
    END_IF;

    // Look at the shift over master distance option to determine profile base type
    IF _I_HmiAxisReq.shiftOverMasterDistance THEN
      // We want to perform the shift over a specified master distance
      _I_Axis.CouplingParameters.ShiftProfileBase := mcPROFBASE_MASTER_DISTANCE;
    ELSE
      // We want to perform the shift based on the master speed and position at the time the shift was triggered
      _I_Axis.CouplingParameters.ShiftProfileBase := mcPROFBASE_MASTER_POSITION;
    END_IF;

    // If requesting to shift back to master position, then overwrite the shift amount
    // by the opposite of the axis offset.
    IF _I_HmiAxisReq.offsetShiftToMasterPosReq THEN
      _I_HmiAxisReq.shiftDistance := -1.0 * _I_SlaveAxis.Status.CalculatedPosition1;
      _I_Axis.CouplingParameters.Shift := -1.0 * _I_SlaveAxis.Status.CalculatedPosition1;
    END_IF;

    // All params should be set. Set the request in the coupling structure and clear the hmi reqs
    _I_Axis.CouplingParameters.OffsetShiftReq := TRUE;
    // turn off the offset and phase shift hmi requests
    _I_HmiAxisReq.offsetShiftReq := FALSE;
    _I_HmiAxisReq.offsetShiftToMasterPosReq := FALSE;
    _I_HmiAxisReq.phaseShiftReq := FALSE;
  ELSIF _I_HmiAxisReq.phaseShiftReq THEN
    // New phase shift request
    // The non request specific params in the coupling structure were set above.
    // Here we need to handle request specific stuff

    // Look at the shift type to determine absolute or relative
    // If the request is to shoft to the master position, then use relative
    IF _I_HmiAxisReq.shiftType = 0 THEN
      // relative
      _I_Axis.CouplingParameters.ShiftMode := mcSHIFT_RELATIVE_NO_RESET;
    ELSIF _I_HmiAxisReq.shiftType = 1 THEN
      // absolute
      _I_Axis.CouplingParameters.ShiftMode := mcSHIFT_ABSOLUTE_NO_RESET;
    ELSE // catch-all -- use relative
      _I_Axis.CouplingParameters.ShiftMode := mcSHIFT_RELATIVE_NO_RESET;
    END_IF;

    // Look at the shift over master distance option to determine profile base type
    IF _I_HmiAxisReq.shiftOverMasterDistance THEN
      // We want to perform the shift over a specified master distance
      _I_Axis.CouplingParameters.ShiftProfileBase := mcPROFBASE_MASTER_DISTANCE;
    ELSE
      // We want to perform the shift based on the master speed and position
      _I_Axis.CouplingParameters.ShiftProfileBase := mcPROFBASE_MASTER_POSITION;
    END_IF;

    // All params should be set. Set the request in the coupling structure and clear the hmi reqs
    _I_Axis.CouplingParameters.PhaseShiftReq := TRUE;
    // turn off the offset and phase shift hmi requests
    _I_HmiAxisReq.offsetShiftReq := FALSE;
    _I_HmiAxisReq.phaseShiftReq := FALSE;
  END_IF;

  // Handle home requests
  IF _I_HmiAxisReq.homeSetZeroReq THEN
    fbHomeSeq._I_Enable := TRUE;
    fbHomeSeq._I_Position := 0.0;
  ELSIF _I_HmiAxisReq.homeSetOffsetReq THEN
    fbHomeSeq._I_Enable := TRUE;
    fbHomeSeq._I_Position := _I_HmiAxisReq.homePosition;
  ELSIF _I_HmiAxisReq.homeSetPosReq THEN
    fbHomeSeq._I_Enable := TRUE;
    fbHomeSeq._I_Position := _I_Axis.Status.Position;
  END_IF;

  // call the home seq fb using the same axis reference as was passed in
  fbHomeSeq(_I_Axis := ADR(_I_Axis));

  // Home reqs processed... now clear them
  _I_HmiAxisReq.homeSetZeroReq := FALSE;
  _I_HmiAxisReq.homeSetOffsetReq := FALSE;
  _I_HmiAxisReq.homeSetPosReq := FALSE;

  // Clear the home seq fb enable once fb is done, error or not
  IF fbHomeSeq._O_Done THEN
    fbHomeSeq._I_Enable := FALSE;
  END_IF;

  // For Error Reset, Drive Reset, Enable, Disable, Brake Release, and Stop Reset, pass these thru and reset the req
  // Home requests are handled separately, so are not cleared here
  _I_Axis.Commands.EnableReq := _I_HmiAxisReq.enableReq;
  _I_Axis.Commands.DisableReq := _I_HmiAxisReq.disableReq;
  _I_Axis.Commands.ReleaseBrakeReq := _I_HmiAxisReq.manBrakeRelReq;
  _I_Axis.Commands.ClearReleaseBrakeReq := _I_HmiAxisReq.clearManBrakeRelReq;
  _I_Axis.Commands.StopResetReq := _I_HmiAxisReq.stopResetReq;
  _I_Axis.Commands.ErrorResetReq := _I_HmiAxisReq.errorResetReq;
  _I_Axis.Commands.DriveResetReq := _I_HmiAxisReq.driveResetReq;
  _I_HmiAxisReq.enableReq := FALSE;
  _I_HmiAxisReq.disableReq := FALSE;
  _I_HmiAxisReq.manBrakeRelReq := FALSE;
  _I_HmiAxisReq.clearManBrakeRelReq := FALSE;
  _I_HmiAxisReq.stopResetReq := FALSE;
  _I_HmiAxisReq.errorResetReq := FALSE;
  _I_HmiAxisReq.driveResetReq := FALSE;

END_FUNCTION_BLOCK

// Given an axis structure, set the basic parameter fb Update bit
// if any of the parameters have changed.
// Update the previous values and clear the fb Update bit once the UpdateDone bit is true.
// A change is detected by comparing the .MoveParameters and the .MoveParametersPrev
// member structures for inequality.
// Note that the entire structure is not compared -- only the part that deals with actual
// move parameters getting sent to hte MpAxisBasic fb is used for comparison, while the
// move permissive parts are not considered.
// Note that an update during a Additive Move will change the target position by
// re-adding the distance. In this case, force the distance to zero. For this reason, the
// mapp move parameter structure is also passed in as a reference IO var.
FUNCTION_BLOCK fbUpdateBasicParams
  // Use the OS to control the execution
  // Set the OS once a change is made until the update is done, then clear the OS
  IF NOT updateOS THEN
    // Get the addresses and size up front
    // Get size and addresses if not yet set
    // IF size = 0 THEN
    // start of where we want to consider for updates
    pParamsStart := ADR(_I_Axis.MoveParameters.Direction);
    // end is where the next thing in memory would start. Account for the size of the last thing
    pParamsEnd := ADR(_I_Axis.MoveParameters.AutoTuneParams) + SIZEOF(_I_Axis.MoveParameters.AutoTuneParams);
    // size is the difference between start and end
    size:= pParamsEnd - pParamsStart;
    // previous values should start at the same element as the current values
    pParamsPrev := ADR(_I_Axis.MoveParametersPrev.Direction);
    // END_IF;

    // See if the member structures are the same. Result will be 0 if they are the same.
    result := brsmemcmp(pParamsPrev,pParamsStart,size);
    IF result <> 0 THEN
      // A parameter change has been made.
      // Set the OS -- we don't need to check or copy memory again until update is done.
      updateOS := TRUE;
      // The fb update bit needs to be set. BUT NOTE: The move additive
      // case is a special case: If a move additive is being executed
      // when an update occurs, the distance is again added to the target
      // position, and the result will be the axis will move past the
      // original target.  Moving to a different place than the original move
      // is probably not what is the operator expects if all they change is
      // velocity or accel/decel for example.  If the distance has changed, while
      // a move additive is active, use the difference in position. This also
      // covers the case where the distance does not change -- delta will be zero.
      IF _I_Axis.Status.IsMoveActive AND
         _I_Axis.Status.AxisDiagnostics.ExecutingCommand = mcAXIS_CMD_MOVE_ADDITIVE THEN
        // A move additive move is being executed, a parameter change is made. The distance
        // parameter is used additively, so use the delta between the new valeu and the old one.
        _IO_MpParams.Distance := _I_Axis.MoveParameters.Distance - _I_Axis.MoveParametersPrev.Distance;
      END_IF;
      _I_Axis.fbMpAxisBasic.Update := TRUE;
    END_IF;
  ELSIF updateOS THEN
    // If the OS is high, an update has at least been requested.  Now look for
    // the update done bit. Update the previous values and clear the update and
    // OS once the done bit is high. Keep the previous value until the end in case
    // their values are helpful during the update.
    IF _I_Axis.fbMpAxisBasic.UpdateDone THEN
      // Update is done. Update the previous values, and clear the request and OS.
      nxtAddr := brsmemcpy(pParamsPrev,pParamsStart,size);
      _I_Axis.fbMpAxisBasic.Update := FALSE;
      updateOS := FALSE;
    END_IF;
  END_IF;
END_FUNCTION_BLOCK

// Calcualte the encoder offset needed for absolute home mode
FUNCTION fctCalcAbsHomeOffset
  fctCalcAbsHomeOffset := _I_DesiredPos - _I_CurrentPos + _I_SetZeroOffset;
END_FUNCTION

// Check CamIn params for a change. Return a boolean, TRUE on no change (equal), FALSE on change (not equal)
FUNCTION fctCheckEqCamInParams
    // This will test the cam in section for equality against the previous values.

    // First check the cam in section
    // Get the start of the gear in params where we want to consider for updates
    pParamsStart := ADR(_I_ParamsA._beginCamInSection);
    // end is where the next thing in memory would start, in this case the end of the section boundary
    pParamsEnd := ADR(_I_ParamsA._endCamInSection);
    // size is the difference between start and end
    size:= pParamsEnd - pParamsStart;
    // previous values should start at the same element as the current values. The previous values are the
    // same structure type, so the name of the starting element and the length are reused
    pParamsPrev := ADR(_I_ParamsB._beginCamInSection);

    // See if the member structures are the same. Result will be 0 if they are the same.
    result := brsmemcmp(pParamsPrev,pParamsStart,size);

    // If parameter change has been detected, return false.
    fctCheckEqCamInParams := (result = 0);

END_FUNCTION

// Check GearIn params for a change. Return a boolean, TRUE on no change (equal), FALSE on change (not equal)
FUNCTION fctCheckEqGearInParams
    // This will test the gear in section and the shift common section for equality
    // against the previous values.

    // First check the gear in section
    // Get the start of the gear in params where we want to consider for updates
    pParamsStart := ADR(_I_ParamsA._beginGearInSection);
    // end is where the next thing in memory would start, in this case the end of the section boundary
    pParamsEnd := ADR(_I_ParamsA._endGearInSection);
    // size is the difference between start and end
    size:= pParamsEnd - pParamsStart;
    // previous values should start at the same element as the current values. The previous values are the
    // same structure type, so the name of the starting element and the length are reused
    pParamsPrev := ADR(_I_ParamsB._beginGearInSection);

    // See if the member structures are the same. Result will be 0 if they are the same.
    result := brsmemcmp(pParamsPrev,pParamsStart,size);
    // If parameter change has been detected, return  false, and no need to go any further.
    // Otherwise check the shift common section
    IF result <> 0 THEN
      fctCheckEqGearInParams := FALSE;
      RETURN;
    ELSE
      // If we get here, the first check was equal.
      // Get the start of the shift common params where we want to consider for updates
       pParamsStart := ADR(_I_ParamsA._beginShiftCommonSection);
      // end is where the next thing in memory would start, in this case the end of the section boundary
      pParamsEnd := ADR(_I_ParamsA._endShiftCommonSection);
      // size is the difference between start and end
      size:= pParamsEnd - pParamsStart;
      // previous values should start at the same element as the current values. The previous values are the
      // same structure type, so the name of the starting element and the length are reused
      pParamsPrev := ADR(_I_ParamsB._beginShiftCommonSection);

      // See if the member structures are the same. Result will be 0 if they are the same.
      result := brsmemcmp(pParamsPrev,pParamsStart,size);
    END_IF;

    // The first check was equal, and this section checks the second section. If the result is zero,
    // no change is detected, and the params are equal.
    fctCheckEqGearInParams := (result = 0);

END_FUNCTION

// Check two move param structures for equality and return a boolean
FUNCTION fctCheckEqMoveParams
  // Use the minimum size -- should be the becuase the two inputs are the same type
  // Check for safety just in case the types change in the future
  size := MIN(SIZEOF(_I_ParamsA),SIZEOF(_I_ParamsB));
  // brsmemcmp returns 0 on equal and < or > 0 when not equal.
  result := brsmemcmp(ADR(_I_ParamsA), ADR(_I_ParamsB), size);
  // Return true on equal, false otherwise
  fctCheckEqMoveParams := (result = 0);
END_FUNCTION

// Check Shift params for a change. Return a boolean, TRUE on no change (equal), FALSE on change (not equal)
FUNCTION fctCheckEqShiftParams
    // This will test the shift and the shift common sections for equality
    // against the previous values.

    // First check the shift section
    // Get the start of the gear in params where we want to consider for updates
    pParamsStart := ADR(_I_ParamsA._beginShiftSection);
    // end is where the next thing in memory would start, in this case the end of the section boundary
    pParamsEnd := ADR(_I_ParamsA._endShiftSection);
    // size is the difference between start and end
    size:= pParamsEnd - pParamsStart;
    // previous values should start at the same element as the current values. The previous values are the
    // same structure type, so the name of the starting element and the length are reused
    pParamsPrev := ADR(_I_ParamsB._beginShiftSection);

    // See if the member structures are the same. Result will be 0 if they are the same.
    result := brsmemcmp(pParamsPrev,pParamsStart,size);
    // If parameter change has been detected, return  false, and no need to go any further.
    // Otherwise check the shift common section
    IF result <> 0 THEN
      fctCheckEqShiftParams := FALSE;
      RETURN;
    ELSE
      // If we get here, the first check was equal.
      // Get the start of the shift common params where we want to consider for updates
       pParamsStart := ADR(_I_ParamsA._beginShiftCommonSection);
      // end is where the next thing in memory would start, in this case the end of the section boundary
      pParamsEnd := ADR(_I_ParamsA._endShiftCommonSection);
      // size is the difference between start and end
      size:= pParamsEnd - pParamsStart;
      // previous values should start at the same element as the current values. The previous values are the
      // same structure type, so the name of the starting element and the length are reused
      pParamsPrev := ADR(_I_ParamsB._beginShiftCommonSection);

      // See if the member structures are the same. Result will be 0 if they are the same.
      result := brsmemcmp(pParamsPrev,pParamsStart,size);
    END_IF;

    // The first check was equal, and this section checks the second section. If the result is zero,
    // no change is detected, and the params are equal.
    fctCheckEqShiftParams := (result = 0);

END_FUNCTION

// Clear command bits in the _IO_sMot_Command parameter if the bit in the eMOT_AXIS_CMD_MASK input mask is clear
FUNCTION fctClearMotionCommands
  // For each command, clear the command if the mask AND comes out clear
  // i.e. Set the bit in the mask to leave the command bit unaltered.
  IF (_I_CmdMask AND MACM_ENABLE_MASK) = 16#0 THEN
    _IO_Commands.EnableCmd := FALSE;
  END_IF;

  IF (_I_CmdMask AND MACM_RELEASE_BRAKE_MASK) = 16#0 THEN
    _IO_Commands.ReleaseBrakeCmd := FALSE;
  END_IF;

  IF (_I_CmdMask AND MACM_HOME_MASK) = 16#0 THEN
    _IO_Commands.HomeCmd := FALSE;
  END_IF;

  IF (_I_CmdMask AND MACM_JOG_MASK) = 16#0 THEN
    _IO_Commands.MoveJogCmd := FALSE;
  END_IF;

  IF (_I_CmdMask AND MACM_JOG_POSITIVE_MASK) = 16#0 THEN
    _IO_Commands.MoveJogPositiveCmd := FALSE;
  END_IF;

  IF (_I_CmdMask AND MACM_JOG_NEGATIVE_MASK) = 16#0 THEN
    _IO_Commands.MoveJogNegativeCmd := FALSE;
  END_IF;

  IF (_I_CmdMask AND MACM_VELOCITY_MOVE_MASK) = 16#0 THEN
    _IO_Commands.MoveVelocityCmd := FALSE;
  END_IF;

  IF (_I_CmdMask AND MACM_RELATIVE_MOVE_MASK) = 16#0 THEN
    _IO_Commands.MoveRelativeCmd := FALSE;
  END_IF;

  IF (_I_CmdMask AND MACM_ABSOLUTE_MOVE_MASK) = 16#0 THEN
    _IO_Commands.MoveAbsoluteCmd := FALSE;
  END_IF;
  (* Slave commands are now in coupling parameters and handled differently
  IF (_I_CmdMask AND MACM_ENGAGE_SLAVE_MASK) = 16#0 THEN
    _IO_Commands.EngageSlaveCmd := FALSE;
  END_IF;

  IF (_I_CmdMask AND MACM_DISENGAGE_SLAVE_MASK) = 16#0 THEN
    _IO_Commands.DisengageSlaveCmd := FALSE;
  END_IF;
  *)
  IF (_I_CmdMask AND MACM_STOP_MASK) = 16#0 THEN
    _IO_Commands.StopCmd := FALSE;
  END_IF;

  IF (_I_CmdMask AND MACM_HALT_MASK) = 16#0 THEN
    _IO_Commands.HaltCmd := FALSE;
  END_IF;

  IF (_I_CmdMask AND MACM_DRIVE_RESET_MASK) = 16#0 THEN
    _IO_Commands.DriveResetCmd := FALSE;
  END_IF;

  // avoid warning for undefined return
  fctClearMotionCommands := TRUE;
END_FUNCTION

// Clear request bits in the _IO_sMot_Command parameter if the bit in the eMOT_AXIS_CMD_MASK input mask is clear
FUNCTION fctClearMotionRequests
  // For each request, clear the request if the mask AND comes out clear
  // i.e. Set the bit in the mask to leave the request bit unaltered.
  IF (_I_ReqMask AND MACM_ENABLE_MASK) = 16#0 THEN
    _IO_Commands.EnableReq := FALSE;
  END_IF;

  IF (_I_ReqMask AND MACM_DISABLE_MASK) = 16#0 THEN
    _IO_Commands.DisableReq := FALSE;
  END_IF;

  IF (_I_ReqMask AND MACM_RELEASE_BRAKE_MASK) = 16#0 THEN
    _IO_Commands.ReleaseBrakeReq := FALSE;
    _IO_Commands.ClearReleaseBrakeReq := FALSE;
  END_IF;

  IF (_I_ReqMask AND MACM_HOME_MASK) = 16#0 THEN
    _IO_Commands.HomeReq := FALSE;
  END_IF;

  IF (_I_ReqMask AND MACM_JOG_MASK) = 16#0 THEN
    _IO_Commands.MoveJogReq := FALSE;
  END_IF;

  IF (_I_ReqMask AND MACM_JOG_POSITIVE_MASK) = 16#0 THEN
    _IO_Commands.MoveJogPositiveReq := FALSE;
  END_IF;

  IF (_I_ReqMask AND MACM_JOG_NEGATIVE_MASK) = 16#0 THEN
    _IO_Commands.MoveJogNegativeReq := FALSE;
  END_IF;

  IF (_I_ReqMask AND MACM_VELOCITY_MOVE_MASK) = 16#0 THEN
    _IO_Commands.MoveVelocityReq := FALSE;
  END_IF;

  IF (_I_ReqMask AND MACM_RELATIVE_MOVE_MASK) = 16#0 THEN
    _IO_Commands.MoveRelativeReq := FALSE;
  END_IF;

  IF (_I_ReqMask AND MACM_ABSOLUTE_MOVE_MASK) = 16#0 THEN
    _IO_Commands.MoveAbsoluteReq := FALSE;
  END_IF;
  (* Slave commands are now in coupling parameters and handled differently
  IF (_I_ReqMask AND MACM_ENGAGE_SLAVE_MASK) = 16#0 THEN
    _IO_Commands.EngageSlaveReq := FALSE;
  END_IF;

  IF (_I_ReqMask AND MACM_DISENGAGE_SLAVE_MASK) = 16#0 THEN
    _IO_Commands.DisengageSlaveReq := FALSE;
  END_IF;
  *)
  IF (_I_ReqMask AND MACM_STOP_MASK) = 16#0 THEN
    _IO_Commands.StopReq := FALSE;
  END_IF;

  IF (_I_ReqMask AND MACM_STOP_RESET_MASK) = 16#0 THEN
    _IO_Commands.StopResetReq := FALSE;
  END_IF;

  IF (_I_ReqMask AND MACM_HALT_MASK) = 16#0 THEN
    _IO_Commands.HaltReq := FALSE;
  END_IF;

  IF (_I_ReqMask AND MACM_DRIVE_RESET_MASK) = 16#0 THEN
    _IO_Commands.DriveResetReq := FALSE;
  END_IF;

  IF (_I_ReqMask AND MACM_ERROR_RESET_MASK) = 16#0 THEN
    _IO_Commands.ErrorResetReq := FALSE;
  END_IF;

  // avoid warning for undefined return
  fctClearMotionRequests := TRUE;

END_FUNCTION

FUNCTION fctCopyAxisStatus
  // Get the addresses and size -- src and dest are the same data type,
  // so no need to check both and take the minimum
  (*
  pParams := ADR(_I_DestStatus);
  pParamsPrev := ADR(_I_Axis.MoveParametersPrev);
  size:= SIZEOF(_I_DestStatus);
*)
  // memcpy(pDest, PSrc, Size)
  nxtAddr := brsmemcpy(ADR(_I_DestStatus),ADR(_I_SrcStatus),SIZEOF(_I_DestStatus));
  fctCopyAxisStatus := TRUE;
END_FUNCTION

// Pack values stored in a MpAxisBasicInfoType structure into a sMot_AxisStatus structure
FUNCTION fctGetMpAxisInfo
  // This provides some flexability and opportunity for conversion/manipulation when using the sMot_AxisStatus
  _IO_UdtStatus.IsCommuncationReady := _I_MpInfo.CommunicationReady;
  _IO_UdtStatus.IsReadyToPowerOn := _I_MpInfo.ReadyToPowerOn;
  _IO_UdtStatus.IsInSimulation := _I_MpInfo.Simulation;
  _IO_UdtStatus.IsJogging := _I_MpInfo.Jogging;
  _IO_UdtStatus.IsAtJogLimit := _I_MpInfo.JogLimitReached;
  _IO_UdtStatus.IsAtTorqueLimit := _I_MpInfo.LimitLoadActive;
  _IO_UdtStatus.PlcOpenState := _I_MpInfo.PLCopenState;
  _IO_UdtStatus.IsAtHomingSwitch := _I_MpInfo.DigitalInputsStatus.HomingSwitch;
  _IO_UdtStatus.IsAtPositiveLimitSwitch := _I_MpInfo.DigitalInputsStatus.PositiveLimitSwitch;
  _IO_UdtStatus.IsAtNegativeLimitSwitch := _I_MpInfo.DigitalInputsStatus.NegativeLimitSwitch;
  _IO_UdtStatus.IsTrigger1Active := _I_MpInfo.DigitalInputsStatus.Trigger1;
  _IO_UdtStatus.IsTrigger2Active := _I_MpInfo.DigitalInputsStatus.Trigger2;
  _IO_UdtStatus.IsDriveEnableActive := _I_MpInfo.DigitalInputsStatus.DriveEnable;
  _IO_UdtStatus.AxisDiagnostics := _I_MpInfo.Diag;
  _IO_UdtStatus.LibraryInfo := _I_MpInfo.LibraryInfo;
  _IO_UdtStatus.networkCommState := _I_MpInfo.CommunicationState;
  _IO_UdtStatus.IsAutoTuneDone := _I_MpInfo.AutoTuneDone;
  _IO_UdtStatus.AutoTuneQuality := _I_MpInfo.AutoTuneQuality;
  _IO_UdtStatus.StartupCount := _I_MpInfo.StartupCount;
  // avoid warning for undefined return
  fctGetMpAxisInfo := TRUE;
END_FUNCTION

// Pack values stored in a sMot_MoveParameter structure into a MpAxisBasicParType structure
FUNCTION fctPackMpAxisBasicParams
  // This provides some flexability and opportunity for conversion/manipulation when using the sMot_MoveParameter
  _IO_MpParams.Position := _I_UdtParams.Position;
  _IO_MpParams.Distance := _I_UdtParams.Distance;
  _IO_MpParams.Velocity := _I_UdtParams.Velocity;
  _IO_MpParams.Acceleration := _I_UdtParams.Acceleration;
  _IO_MpParams.Deceleration := _I_UdtParams.Deceleration;
  _IO_MpParams.Direction := _I_UdtParams.Direction;
  _IO_MpParams.Homing := _I_UdtParams.HomeParams;
  _IO_MpParams.Jog := _I_UdtParams.JogParams;
  _IO_MpParams.Stop := _I_UdtParams.StopParams;
  _IO_MpParams.LimitLoad := _I_UdtParams.TorqueLimitParams;
  _IO_MpParams.AutoTune := _I_UdtParams.AutoTuneParams;
  _IO_MpParams.Jerk := _I_UdtParams.MaxJerk;
  // avoid warning for undefined return
  fctPackMpAxisBasicParams := TRUE;
END_FUNCTION
```

### Library Logical/Libraries/GAConvert (IEC)

#### GAConvert.var - Exported constants
```iecst
(********************************************************************
 * COPYRIGHT -- General Atomics
 ********************************************************************
 * Library: GAConvert
 * File: GAConvert.var
 * Author: Administrator
 * Created: November 03, 2013
 ********************************************************************
 * Constants of library GAConvert
 ********************************************************************)

VAR CONSTANT
  B_MASKALL_SET   : BYTE   := 16#FF;
  B_MASKBIT00_SET : BYTE  := 16#01;
  B_MASKBIT01_SET : BYTE  := 16#02;
  B_MASKBIT02_SET : BYTE  := 16#04;
  B_MASKBIT03_SET : BYTE  := 16#08;
  B_MASKBIT04_SET : BYTE  := 16#10;
  B_MASKBIT05_SET : BYTE  := 16#20;
  B_MASKBIT06_SET : BYTE  := 16#40;
  B_MASKBIT07_SET : BYTE  := 16#80;

  B_MASKALL_CLEAR   : BYTE  := 16#00;
  B_MASKBIT00_CLEAR : BYTE  := 16#FE;
  B_MASKBIT01_CLEAR : BYTE  := 16#FD;
  B_MASKBIT02_CLEAR : BYTE  := 16#FB;
  B_MASKBIT03_CLEAR : BYTE  := 16#F7;
  B_MASKBIT04_CLEAR : BYTE  := 16#EF;
  B_MASKBIT05_CLEAR : BYTE  := 16#EF;
  B_MASKBIT06_CLEAR : BYTE  := 16#BF;
  B_MASKBIT07_CLEAR : BYTE  := 16#7F;

  W_MASKALL_SET   : WORD   := 16#FFFF;
  W_MASKBIT00_SET : WORD  := 16#01;
  W_MASKBIT01_SET : WORD  := 16#02;
  W_MASKBIT02_SET : WORD  := 16#04;
  W_MASKBIT03_SET : WORD  := 16#08;
  W_MASKBIT04_SET : WORD  := 16#10;
  W_MASKBIT05_SET : WORD  := 16#20;
  W_MASKBIT06_SET : WORD  := 16#40;
  W_MASKBIT07_SET : WORD  := 16#80;
  W_MASKBIT08_SET : WORD  := 16#100;
  W_MASKBIT09_SET : WORD  := 16#200;
  W_MASKBIT10_SET : WORD := 16#400;
  W_MASKBIT11_SET : WORD := 16#800;
  W_MASKBIT12_SET : WORD := 16#1000;
  W_MASKBIT13_SET : WORD := 16#2000;
  W_MASKBIT14_SET : WORD := 16#4000;
  W_MASKBIT15_SET : WORD := 16#8000;

  W_MASKALL_CLEAR   : WORD   := 16#0;
  W_MASKBIT00_CLEAR : WORD  := 16#FFFE;
  W_MASKBIT01_CLEAR : WORD  := 16#FFFD;
  W_MASKBIT02_CLEAR : WORD  := 16#FFFB;
  W_MASKBIT03_CLEAR : WORD  := 16#FFF7;
  W_MASKBIT04_CLEAR : WORD  := 16#FFEF;
  W_MASKBIT05_CLEAR : WORD  := 16#FFEF;
  W_MASKBIT06_CLEAR : WORD  := 16#FFBF;
  W_MASKBIT07_CLEAR : WORD  := 16#FF7F;
  W_MASKBIT08_CLEAR : WORD  := 16#FEFF;
  W_MASKBIT09_CLEAR : WORD  := 16#FDFF;
  W_MASKBIT10_CLEAR : WORD := 16#FBFF;
  W_MASKBIT11_CLEAR : WORD := 16#F7FF;
  W_MASKBIT12_CLEAR : WORD := 16#EFFF;
  W_MASKBIT13_CLEAR : WORD := 16#DFFF;
  W_MASKBIT14_CLEAR : WORD := 16#BFFF;
  W_MASKBIT15_CLEAR : WORD := 16#7FFF;

  DW_MASKALL_SET   : DWORD   := 16#FFFFFFFF;
  DW_MASKBIT00_SET : DWORD  := 16#01;
  DW_MASKBIT01_SET : DWORD  := 16#02;
  DW_MASKBIT02_SET : DWORD  := 16#04;
  DW_MASKBIT03_SET : DWORD  := 16#08;
  DW_MASKBIT04_SET : DWORD  := 16#10;
  DW_MASKBIT05_SET : DWORD  := 16#20;
  DW_MASKBIT06_SET : DWORD  := 16#40;
  DW_MASKBIT07_SET : DWORD  := 16#80;
  DW_MASKBIT08_SET : DWORD  := 16#100;
  DW_MASKBIT09_SET : DWORD  := 16#200;
  DW_MASKBIT10_SET : DWORD := 16#400;
  DW_MASKBIT11_SET : DWORD := 16#800;
  DW_MASKBIT12_SET : DWORD := 16#1000;
  DW_MASKBIT13_SET : DWORD := 16#2000;
  DW_MASKBIT14_SET : DWORD := 16#4000;
  DW_MASKBIT15_SET : DWORD := 16#8000;
  DW_MASKBIT16_SET : DWORD := 16#10000;
  DW_MASKBIT17_SET : DWORD := 16#20000;
  DW_MASKBIT18_SET : DWORD := 16#40000;
  DW_MASKBIT19_SET : DWORD := 16#80000;
  DW_MASKBIT20_SET : DWORD := 16#100000;
  DW_MASKBIT21_SET : DWORD := 16#200000;
  DW_MASKBIT22_SET : DWORD := 16#400000;
  DW_MASKBIT23_SET : DWORD := 16#800000;
  DW_MASKBIT24_SET : DWORD := 16#1000000;
  DW_MASKBIT25_SET : DWORD := 16#2000000;
  DW_MASKBIT26_SET : DWORD := 16#4000000;
  DW_MASKBIT27_SET : DWORD := 16#8000000;
  DW_MASKBIT28_SET : DWORD := 16#10000000;
  DW_MASKBIT29_SET : DWORD := 16#20000000;
  DW_MASKBIT30_SET : DWORD := 16#40000000;
  DW_MASKBIT31_SET : DWORD := 16#80000000;

  DW_MASKALL_CLEAR   : DWORD   := 16#0;
  DW_MASKBIT00_CLEAR : DWORD  := 16#FFFFFFFE;
  DW_MASKBIT01_CLEAR : DWORD  := 16#FFFFFFFD;
  DW_MASKBIT02_CLEAR : DWORD  := 16#FFFFFFFB;
  DW_MASKBIT03_CLEAR : DWORD  := 16#FFFFFFF7;
  DW_MASKBIT04_CLEAR : DWORD  := 16#FFFFFFEF;
  DW_MASKBIT05_CLEAR : DWORD  := 16#FFFFFFEF;
  DW_MASKBIT06_CLEAR : DWORD  := 16#FFFFFFBF;
  DW_MASKBIT07_CLEAR : DWORD  := 16#FFFFFF7F;
  DW_MASKBIT08_CLEAR : DWORD  := 16#FFFFFEFF;
  DW_MASKBIT09_CLEAR : DWORD  := 16#FFFFFDFF;
  DW_MASKBIT10_CLEAR : DWORD := 16#FFFFFBFF;
  DW_MASKBIT11_CLEAR : DWORD := 16#FFFFF7FF;
  DW_MASKBIT12_CLEAR : DWORD := 16#FFFFEFFF;
  DW_MASKBIT13_CLEAR : DWORD := 16#FFFFDFFF;
  DW_MASKBIT14_CLEAR : DWORD := 16#FFFFBFFF;
  DW_MASKBIT15_CLEAR : DWORD := 16#FFFF7FFF;
  DW_MASKBIT16_CLEAR : DWORD := 16#FFFEFFFF;
  DW_MASKBIT17_CLEAR : DWORD := 16#FFFDFFFF;
  DW_MASKBIT18_CLEAR : DWORD := 16#FFFBFFFF;
  DW_MASKBIT19_CLEAR : DWORD := 16#FFF7FFFF;
  DW_MASKBIT20_CLEAR : DWORD := 16#FFEFFFFF;
  DW_MASKBIT21_CLEAR : DWORD := 16#FFDFFFFF;
  DW_MASKBIT22_CLEAR : DWORD := 16#FFBFFFFF;
  DW_MASKBIT23_CLEAR : DWORD := 16#FF7FFFFF;
  DW_MASKBIT24_CLEAR : DWORD := 16#FEFFFFFF;
  DW_MASKBIT25_CLEAR : DWORD := 16#FDFFFFFF;
  DW_MASKBIT26_CLEAR : DWORD := 16#FBFFFFFF;
  DW_MASKBIT27_CLEAR : DWORD := 16#F7FFFFFF;
  DW_MASKBIT28_CLEAR : DWORD := 16#EFFFFFFF;
  DW_MASKBIT29_CLEAR : DWORD := 16#DFFFFFFF;
  DW_MASKBIT30_CLEAR : DWORD := 16#BFFFFFFF;
  DW_MASKBIT31_CLEAR : DWORD := 16#7FFFFFFF;

END_VAR
```

#### GAConvert.fun - Exported functions and function blocks
```iecst
(********************************************************************
 * COPYRIGHT -- General Atomics
 ********************************************************************
 * Library: GAConvert
 * File: GAConvert.fun
 * Author: Administrator
 * Created: November 03, 2013
 ********************************************************************
 * Functions and function blocks of library GAConvert
 ********************************************************************)

FUNCTION USINT2_TO_UINT : UINT (* Pack two USINTs into a UINT and return the UINT *)
  VAR_INPUT
    src0 : USINT; (* USINT to be converted to lower order byte of UINT *)
    src1 : USINT; (* USINT to be converted to higher order byte of UINT *)
  END_VAR
END_FUNCTION

FUNCTION USINT4_TO_UDINT : UDINT (* Pack 4 USINTs into a UDINT and return the UDINT *)
  VAR_INPUT
    src0 : USINT; (* USINT to be converted to lower order byte of UDINT *)
    src1 : USINT; (* USINT to be converted to second byte of UDINT *)
    src2 : USINT; (* USINT to be converted to third byte of UDINT *)
    src3 : USINT; (* USINT to be converted to highest order byte of UDINT *)
  END_VAR
  VAR
    tempUDINT1 : UDINT; (* temporary holding spot *)
    tempUDINT2 : UDINT; (* temporary holding spot *)
  END_VAR
END_FUNCTION

FUNCTION UINT_TO_2USINT : BOOL (* Split UINT to two USINTs *)
	VAR_INPUT
		src_int : UINT; (* input int which gets divided into two bytes *)
	END_VAR
	VAR_IN_OUT
		dest0 : USINT; (* lower byte of UINT *)
		dest1 : USINT; (* upper byte of UINT *)
	END_VAR
END_FUNCTION

FUNCTION AxisIndex_To_ColPairIndex : DINT (* Convert an axis index 1-24 to column pair index 1-6 and return the colum pair index *)
  VAR_INPUT
    axisIndex : DINT;
  END_VAR
  VAR
    tempIndex : DINT;
  END_VAR
END_FUNCTION
```

#### GAConvert.st - Implementation code
```iecst
(********************************************************************
 * COPYRIGHT -- General Atomics
 ********************************************************************
 * Program: HBConvert
 * File: HBConvert.st
 * Author: Administrator
 * Created: November 03, 2013
 ********************************************************************
 * Implementation of program HBConvert
 ********************************************************************)

(* Split a UINT into two USINTs *)
FUNCTION UINT_TO_2USINT // Return bool true always
  //	VAR_INPUT
  //		src_int : UINT; (* input int which gets divided into two bytes *)
  //	END_VAR
  //	VAR_IN_OUT
  //		dest0 : USINT; (* lower byte of UINT *)
  //		dest1 : USINT; (* upper byte of UINT *)
  //	END_VAR

	dest0:= UINT_TO_USINT(src_int);
	dest1:= UINT_TO_USINT(SHR(src_int, 8));
	UINT_TO_2USINT:= TRUE; // always return true
END_FUNCTION

 (* Pack two USINTs into a UINT and return the UINT *)
FUNCTION USINT2_TO_UINT // return a UINT
  //	VAR_INPUT
  //		src0 : USINT; (* USINT to be converted to lower order byte of UINT *)
  //		src1 : USINT; (* USINT to be converted to higher order byte of UINT *)
  //	END_VAR

	// shift hi byte up by 8, and OR with low byte
	USINT2_TO_UINT:= SHL(USINT_TO_UINT(src1),8) OR src0;
END_FUNCTION

 (* Pack 4 USINTs into a UDINT and return the UDINT *)
FUNCTION USINT4_TO_UDINT  // Return UDINT
  //	VAR_INPUT
  //		src0 : USINT; (* USINT to be converted to lower order byte of UDINT *)
  //		src1 : USINT; (* USINT to be converted to second byte of UDINT *)
  //		src2 : USINT; (* USINT to be converted to third byte of UDINT *)
  //		src3 : USINT; (* USINT to be converted to highest order byte of UDINT *)
  //	END_VAR

	// shift hi byte up by 24 and next byte up by 16
	tempUDINT1:= SHL(USINT_TO_UDINT(src1), 8) OR src0; // lower two bytes
	tempUDINT2:= SHL(USINT_TO_UDINT(src3), 24) OR SHL(USINT_TO_UDINT(src2), 16); // hightest two bytes
  USINT4_TO_UDINT:= tempUDINT1 OR tempUDINT2;
END_FUNCTION

(* Convert an axis index 1-24 to a column pair index 1-6 *)
(* if foot index is outside the 1-24 range, return 0 *)
FUNCTION AxisIndex_To_ColPairIndex  // return DINT
//  VAR_INPUT
//    axisIndex : DINT;
//  END_VAR

// axis index 1, 2, 13, or 14 return colum pair index 1
// axis index 3, 4, 15, or 16 return column pair index 2
// axis index 5, 6, 17, or 18 return column pair index 3
// axis index 7, 8, 19, or 29 return column pair index 4
// axis index 9, 10, 21, or 22 return column pair index 5
// axis index 11, 12, 23, or 24 return column pair index 6

  // if the axis index is 1-12 (a foot) then the column pair index is = (foot index + foot index mod 2) / 2
  // if the axis index is 13-24 (a column) then the colum pair is the same as above, but first subtract 12 from the axis index
  IF axisIndex >= 1 AND axisIndex <= 12 THEN
    // axis index is a foot
    AxisIndex_To_ColPairIndex:= (axisIndex + (axisIndex MOD 2)) / 2;
  ELSIF axisIndex > 12 AND axisIndex <= 24 THEN
    // axis index is a column
    tempIndex:= axisIndex - 12;
    AxisIndex_To_ColPairIndex:= (tempIndex + (tempIndex MOD 2)) / 2;
  ELSE
    // axis index is invalid
    AxisIndex_To_ColPairIndex:= 0;
  END_IF;

END_FUNCTION
```

### Library Logical/Libraries/GAMath (IEC)

#### GAMath.fun
```iecst
(********************************************************************
 * COPYRIGHT -- General Atomics
 ********************************************************************
 * Library: GAMath
 * File: GAMathj.fun
 * Author: J Sheeron
 ********************************************************************
 * Functions and function blocks of library GAMath
 ********************************************************************)

FUNCTION_BLOCK fbCalcTrapMoveTime
  VAR_INPUT
    _I_Vel0 : REAL := 0.0; (* units/sec starting velocity *)
    _I_VelMove : REAL; (* units/sec desired move velocity*)
    _I_Accel : REAL; (* untis/sec^2 *)
    _I_Decel : REAL; (* untis/sec^2 *)
    _I_Dist : LREAL; (* units, LREAL to be compatible with motion system *)
  END_VAR

  VAR_OUTPUT
    _O_MoveTime : TIME; (* how long will the move take as a TIME type *)
    _O_MoveTimeMsec : DINT; (* mSec, how long the move will take *)
    _O_VelReached : REAL; (* units/sec. Velocity reached will be <= VelMove for triangular profiles, dist < Dcheck *)
    _O_Dcheck : LREAL; (* units. Distances > than this have a trapazoidal shape and VelReached = VelMove *)
  END_VAR

  VAR
    v0 : REAL; (* internal copy of input *)
    vMove : REAL; (* internal copy of input *)
    accel : REAL; (* internal copy of input *)
    decel : REAL; (* internal copy of input *)
    dist : LREAL; (* internal copy of input *)
    tval1  : LREAL; (* temporary value *)
    tval2  : LREAL; (* temporary value *)
    tval3  : LREAL; (* temporary value *)
    tval4  : LREAL; (* temporary value *)
    tval5  : LREAL; (* temporary value *)
    seconds : LREAL; (* temporary value *)
  END_VAR
END_FUNCTION_BLOCK

FUNCTION_BLOCK fbLookUpYValT3 (* Given an X, get the Y value. Interpolate if needed. *)
	VAR CONSTANT
		INVALID_SENTINEL : REAL := -9999.0;
	END_VAR

	VAR_INPUT
    LoadTables : BOOL; (* load lookup table values *)
    Enable : BOOL; (* trigger a lookup *)
		XVal : REAL; (* x value to lookup *)
		T1 : REFERENCE TO sXYTableReal50; (* table 1 *)
		T2 : REFERENCE TO sXYTableReal50; (* table 2 *)
		T3 : REFERENCE TO sXYTableReal50; (* table 3 *)
	END_VAR

	VAR_OUTPUT
    IsTablesLoaded : BOOL; (* look up tables have been loaded *)
    Active : BOOL;
    Done : BOOL;
    Error : BOOL;
		YVal : REAL; (* looked up and interpolated Y value *)
	END_VAR

	VAR
    (* oneshots *)
    _loadOS : BOOL := FALSE;
    _enableOS : BOOL := FALSE;
    (* which table to use *)
		_xValPrev : REAL; (* previous x value to lookup *)
    _tableNumber : USINT;
    (* table lookup fbs*)
		_fbDepthToAngleLuT1 : MTLookUpTable;
		_fbDepthToAngleLuT2 : MTLookUpTable;
		_fbDepthToAngleLuT3 : MTLookUpTable;
	END_VAR
END_FUNCTION_BLOCK

FUNCTION fctAziDiff : LREAL (* Return the angle between pos A and pos B (A-B). Returns +/- 180 deg. +: Pos A ahead of B, -: Pos A behind B *)
  (*
  Result is +/- 180 degrees
  Positive value: A is ahead of B.
  Negative value: A is behind B.
  Account for 360 deg rollover. *)
  VAR_INPUT
    _I_PosA : LREAL;
    _I_PosB : LREAL;
  END_VAR

  VAR
    angle : LREAL;
  END_VAR
END_FUNCTION

FUNCTION fctLRCeiling : LREAL (* LREAL Ceiling -- Return the smallest whole number not less than value *)
  VAR_INPUT
    _I_Val : LREAL;
  END_VAR

  VAR
    val1 : LREAL;
    rem : LREAL;
  END_VAR
END_FUNCTION

FUNCTION fctLRFloor : LREAL (* LREAL floor -- Return the largest whole number not greater than value *)
  VAR_INPUT
    _I_Val : LREAL;
  END_VAR

  VAR
    val1 : LREAL;
  END_VAR
END_FUNCTION

FUNCTION fctLRFract : LREAL (* LREAL fractional -- Return the fractional part of a value *)
  VAR_INPUT
    _I_Val : LREAL;
  END_VAR

  VAR
    val1 : LREAL;
  END_VAR
END_FUNCTION

FUNCTION fctLRMod : LREAL (* LREAL MOD -- Return the remainder of Dividend MOD Divisor *)
  VAR_INPUT
    _I_Dividend : LREAL;
    _I_Divisor : LREAL;
  END_VAR

  VAR
    val1 : LREAL;
    rem : LREAL;
  END_VAR
END_FUNCTION

FUNCTION fctRound1 : REAL (* Return the source value (real) rounded to 1 decimal place *)
  VAR_INPUT
    _I_src : LREAL; (* REAL value to be rounded *)
  END_VAR
  VAR
    dintTemp : DINT; (* temp value *)
  END_VAR
END_FUNCTION

FUNCTION fctRound2 : REAL (* Return the source value (real) rounded to 2 decimal places *)
  VAR_INPUT
    _I_src : LREAL; (* REAL value to be rounded *)
  END_VAR
  VAR
    dintTemp : DINT; (* temp value *)
  END_VAR
END_FUNCTION

FUNCTION fctRound3 : REAL (* Return the source value (real) rounded to 2 decimal places *)
  VAR_INPUT
    _I_src : LREAL; (* REAL value to be rounded *)
  END_VAR
  VAR
    dintTemp : DINT; (* temp value *)
  END_VAR
END_FUNCTION

FUNCTION fctLRound1 : LREAL (* Return the source value (LREAL) rounded to 1 decimal place *)
  VAR_INPUT
    _I_src : LREAL; (* REAL value to be rounded *)
  END_VAR
  VAR
    dintTemp : DINT; (* temp value *)
  END_VAR
END_FUNCTION

FUNCTION fctLRound2 : LREAL (* Return the source value (LREAL) rounded to 2 decimal places *)
  VAR_INPUT
    _I_src : LREAL; (* REAL value to be rounded *)
  END_VAR
  VAR
    dintTemp : DINT; (* temp value *)
  END_VAR
END_FUNCTION

FUNCTION fctLRound3 : LREAL (* Return the source value (LREAL) rounded to 2 decimal places *)
  VAR_INPUT
    _I_src : LREAL; (* REAL value to be rounded *)
  END_VAR
  VAR
    dintTemp : DINT; (* temp value *)
  END_VAR
END_FUNCTION

FUNCTION fctSwapTableT3 : USINT (* Swap X & Y columns *)
	VAR_INPUT
		table : REFERENCE TO sXYTableReal50; (* table to swap the X & Y values of *)
	END_VAR
	VAR
		tVals : ARRAY[0..49] OF REAL; (* temporary storage *)
		length : UDINT; (* mem copy length in bytes *)
		nextAddr : UDINT; (* return from memcpy *)
	END_VAR
END_FUNCTION
```
